// Map values
VIR.Position := Position;
VIR.NumOfKeyValuePairs := NumOfKeyValuePairs;
VIR.KeyValuePair := KeyValuePairs;

// Forward to ITC
F_ITC_SendVIR := fbITC_Manager.M_SendData(
					meChannel	:= eChannelSrc,
					mMsgType	:= E_ITC_MsgTypeConv.VISUALIZATION_INFORMATION_REPORT,
					mpData		:= ADR(VIR),
					mLen        := SIZEOF(VIR));

END_FUNCTION

// ---- 20_Product/10_BCF/11_Conv/10_Base/F_SearchPositionOfTU_Index.TcPOU
FUNCTION F_SearchPositionOfTU_Index : ST_PositionIdent
(**************************************************************************************
 * 	Application		:	BoxControl Framework
 *	Revision		:	$Revision: 464436 $
 *	Revision date	:	$Date: 2020-10-27 15:58:44 +0100 (tis, 27 okt 2020) $
 *	Last changed by	:	$Author: d7mangc $
 *	URL				:	$URL: http://almscdc.swisslog.com/repo/SWPD/Development/BoxControlFramework/20_Release/tags/R1.12.0/01_Software/BCF/BCF/JumpStart/20_Product/10_BCF/11_Conv/10_Base/F_SearchPositionOfTU_Index.TcPOU $
 *
 *	Purpose			:	Searchs for the FunctionNumber according the TU-DataIndex.
 *						
 *
 * ------------------------------------------------------------------------------------
 *	Copyright Swisslog [IP AG], Switzerland. All rights reserved.
 * 
 * ------------------------------------------------------------------------------------
 *	
 * 	Revision History: 
 *
 * 	VERSION			DATE			INITIALS			DESCRIPTION
 *	0.1				01.01.2001		swl					Example
 *
 **************************************************************************************)
VAR_INPUT
	TU_DataIndex  			: DINT; // Index variable
	eStartFunctionNumber 	: E_FunctionNumber; // Start loop from this ElementNumber 
END_VAR

VAR
	eFunctionNumber  		: E_FunctionNumber;  // Function incrementor 
	ZoneNumber				: INT; // Zone number
	FoundOnFunction			: BOOL; // Requested index was found on a function
	FoundOnZone				: BOOL; // Requested index was found on a zone
END_VAR

// Initialize
F_SearchPositionOfTU_Index.eFunctionNumber := 0;
F_SearchPositionOfTU_Index.ZoneNumber := 0;

// If no start function number is set
IF eStartFunctionNumber <= 0 THEN
	//Default set first function
	eStartFunctionNumber := F_BEGIN_FUNCTION + 1;
END_IF

// Loop through all functions
FOR eFunctionNumber := eStartFunctionNumber TO F_END_FUNCTION - 1 BY 1 DO
	// If a valid reference was found, check if a function contains on any
	// zone the requested TU Index 
	IF __ISVALIDREF(FunctionRegistry[eFunctionNumber].rFunction) THEN
		FoundOnFunction := FunctionRegistry[eFunctionNumber].rFunction.M_FindTU_DataIndex(
							mZoneNumber := 0,
							mTU_DataIndex := TU_DataIndex);

		// If the requested index could be determined on a function,
		// try to find the specific zone
		IF FoundOnFunction THEN
			// Set return value of the function	
			F_SearchPositionOfTU_Index.eFunctionNumber := eFunctionNumber;
		
			// Loop through all zones of this function 
			FOR ZoneNumber := 1 TO FunctionRegistry[eFunctionNumber].rFunction.SettingsFunction.NumberOfZones BY 1 DO
				FoundOnZone := FunctionRegistry[eFunctionNumber].rFunction.M_FindTU_DataIndex(
								mZoneNumber := ZoneNumber,
								mTU_DataIndex := TU_DataIndex);
				// Zone was found 
				IF FoundOnZone THEN
					// Set return value of the zone
					F_SearchPositionOfTU_Index.ZoneNumber := ZoneNumber;
					EXIT;
				END_IF
			END_FOR
		END_IF
		
		// If search was succesful
		IF FoundOnFunction THEN
			// Stop, and return result
			RETURN;
		END_IF
	END_IF
END_FOR

// Update position name
F_SearchPositionOfTU_Index.PositionName := F_GetFunctionName(eFunctionNumber := F_SearchPositionOfTU_Index.eFunctionNumber,
															 ZoneNumber := F_SearchPositionOfTU_Index.ZoneNumber);

END_FUNCTION

// ---- 20_Product/10_BCF/11_Conv/12_E_Functions/10_Helper/F_GetFunctionName.TcPOU
FUNCTION F_GetFunctionName : STRING(NAME_LENGTH)
(**************************************************************************************
 * 	Application		:	BoxControl Framework
 *	Revision		:	$Revision: 404529 $
 *	Revision date	:	$Date: 2018-04-23 08:21:38 +0200 (Mo., 23 Apr 2018) $
 *	Last changed by	:	$Author: b7bolm $
 *	URL				:	$URL: http://almscdc.swisslog.com/repo/SWPD/Development/BoxControlFramework/20_Release/trunk/01_Software/BCF/BCF/JumpStart/20_Product/10_App/12_E_Functions/10_Lib/10_Conv/10_Functions/F_GetFunctionName.TcPOU $
 *
 *	Purpose			:	Return function name
 *
 * ------------------------------------------------------------------------------------
 *	Copyright Swisslog [IP AG], Switzerland. All rights reserved.
 * 
 * ------------------------------------------------------------------------------------
 *	
 * 	Revision History: 
 *
 * VERSION DATE         INITIALS     DESCRIPTION
 * 0.0     DD.MM.YYYY   (name)       (explain customized modifications)
 *
 **************************************************************************************)
VAR_INPUT
	eFunctionNumber		: E_FunctionNumber; // Function number
	ZoneNumber			: INT; // Zone number
END_VAR
VAR
	DebugMsg				: T_MAXSTRING; // Debug message
END_VAR

// Check if function number is valid
IF eFunctionNumber > E_FunctionNumber.F_BEGIN_FUNCTION AND
   eFunctionNumber < E_FunctionNumber.F_END_FUNCTION THEN

	// Check reference is valid
	IF __ISVALIDREF(FunctionRegistry[eFunctionNumber].rFunction) THEN
		// If the request goes to the function
		IF ZoneNumber = 0 THEN
			// Return function name
			F_GetFunctionName := FunctionRegistry[eFunctionNumber].rFunction.SettingsFunction.FunctionName;
		ELSIF ZoneNumber > 0 AND ZoneNumber <= NUMBER_OF_ZONES_PER_FUNCTION THEN
			// Return zone name
			F_GetFunctionName := FunctionRegistry[eFunctionNumber].rFunction.SettingsFunction.Zone[ZoneNumber].ZoneName;
		ELSE
			F_GetFunctionName:= '';
			//-- debug message ------------------------------------------------
			// example: '11-000-0000-00-0,  invalid function/zone number,  function = 21,  zone = 1'
			DebugMsg:= '';
			DebugMsg:= CONCAT(DebugMsg, F_AddDividerToSisString(SubsystemRegistry.SubsystemName));
			DebugMsg:= CONCAT(DebugMsg, ',  invalid function/zone number');
			DebugMsg:= CONCAT(DebugMsg, DebugTextBlocks.FUNCTIONNBR);
			DebugMsg:= CONCAT(DebugMsg, TO_STRING(eFunctionNumber));
			DebugMsg:= CONCAT(DebugMsg, DebugTextBlocks.ZONENBR);
			DebugMsg:= CONCAT(DebugMsg, INT_TO_STRING(ZoneNumber));
			fbDebugMsgManager.M_SendMessage(meMessageType:= E_DebugMsgType.ERROR,
											mDebugSource := 'F_GetFunctionName', 
											mpMsgData    := ADR(DebugMsg),
											mMsgDataLen  := INT_TO_UDINT(LEN(DebugMsg)));
		END_IF
   END_IF
END_IF

END_FUNCTION

// ---- 20_Product/10_BCF/11_Conv/12_E_Functions/10_Helper/F_AddDividerToSisString.TcPOU
// adds '-' divider to a sis string: MMGGGEEEEFFZ -> MM-GGG-EEEE-FF-Z, even if there is already some dividers: M-M-G-G-G-E-E-E-E-F-F-Z -> MM-GGG-EEEE-FF-Z
FUNCTION PUBLIC F_AddDividerToSisString : STRING[NAME_LENGTH]

(**************************************************************************************
 * 	Application		:	BoxControl Framework
 *	Revision		:	$Revision: 461869 $
 *	Revision date	:	$Date: 2020-09-25 14:40:24 +0200 (Fr., 25 Sep 2020) $
 *	Last changed by	:	$Author: d7mangc $
 *	URL				:	$URL: http://almscdc.swisslog.com/repo/SWPD/Development/BoxControlFramework/20_Release/branches/R1.x/01_Software/BCF/BCF/JumpStart/20_Product/10_BCF/11_Conv/12_E_Functions/10_Helper/F_CreateTU_DataString.TcPOU $
 *
 *	Purpose			:	adds divider between subsystem, switchgroup, element, function and zone number
 * 						String: 'MM-GGG-EEEE-FF-Z'
 *
 * ------------------------------------------------------------------------------------
 *	Copyright Swisslog [IP AG], Switzerland. All rights reserved.
 * 
 * ------------------------------------------------------------------------------------
 *	
 * 	Revision History: 
 *
 * VERSION DATE         INITIALS     DESCRIPTION
 * 0.0     DD.MM.YYYY   (name)       (explain customized modifications)
 *
 **************************************************************************************)

//***********************************************************************************************************
VAR_INPUT
	Name				: STRING[NAME_LENGTH]		:= '';
END_VAR

//***********************************************************************************************************
VAR
	Without				: STRING[NAME_LENGTH]		:= '';
	Result				: STRING[NAME_LENGTH]		:= '';
	Src					: WORD						:= 0;
	Dst					: WORD						:= 0;
	Char				: BYTE						:= 0;
END_VAR


// initialize
memset( destAddr:= ADR(Without),  fillByte:= 16#00,  n:= SIZEOF(Without)  );
memset( destAddr:= ADR(Result),   fillByte:= 16#00,  n:= SIZEOF(Result)   );


// has name already divider? ( and remove it)
Src:= 0;
Dst:= 0;
WHILE(Name[Src] <> 16#00)DO
	Char:= Name[Src];
	Src := Src + 1;

	// valid characters?
	IF(Char >= 16#30) AND (Char <= 16#39)THEN
		Without[Dst]:= Char;
		Dst:= Dst + 1;
		CONTINUE;

	ELSIF Char >= 16#2D THEN (* '-' *)
		CONTINUE;
	END_IF

	// invalid
	F_AddDividerToSisString:= Name;
	RETURN;
END_WHILE


// add divider to specific positions
Src:= 0;
Dst:= 0;
WHILE(Without[Src] <> 16#00)DO
	// string ends
	IF Dst >= SIZEOF(Result) THEN
		Dst:= SIZEOF(Result) - 1; // make space for termination
		EXIT;
	END_IF
	
	// add divider
	IF    Src =  2 THEN  Result[Dst]:= 16#2D;  Dst:= Dst + 1;  // MM -> GGG
	ELSIF Src =  5 THEN  Result[Dst]:= 16#2D;  Dst:= Dst + 1;  // GGG -> EEEE
	ELSIF Src =  9 THEN  Result[Dst]:= 16#2D;  Dst:= Dst + 1;  // EEEE -> FF
	ELSIF Src = 11 THEN  Result[Dst]:= 16#2D;  Dst:= Dst + 1;  // FF -> Z
	END_IF
	
	// string ends
	IF Dst >= SIZEOF(Result)THEN
		Dst:= SIZEOF(Result) - 1; // make space for termination
		EXIT;
	END_IF
	
	// copy character
	Result[Dst]:= Without[Src];
	
	// continue
	Src:= Src + 1;
	Dst:= Dst + 1;
END_WHILE

Result[Dst]:= 16#00;


// done
F_AddDividerToSisString:= Result;

END_FUNCTION

// ---- 20_Product/10_BCF/11_Conv/12_E_Functions/10_Helper/F_CreateTU_DataString.TcPOU
// Creates a text string with TU data information: 'TU_DataIndex = 1979,  TuID = 0012345600,  AssignmentID = 19790109'
FUNCTION PUBLIC F_CreateTU_DataString : STRING[127]

(**************************************************************************************
 * 	Application		:	BoxControl Framework
 *	Revision		:	$Revision: 474106 $
 *	Revision date	:	$Date: 2021-03-26 07:58:15 +0100 (fre, 26 mar 2021) $
 *	Last changed by	:	$Author: d7mangc $
 *	URL				:	$URL: http://almscdc.swisslog.com/repo/SWPD/Development/BoxControlFramework/20_Release/tags/R1.12.0/01_Software/BCF/BCF/JumpStart/20_Product/10_BCF/11_Conv/12_E_Functions/10_Helper/F_CreateTU_DataString.TcPOU $
 *
 *	Purpose			:	Creates a text string with TU data information which can be used for debug messages
 * 						String: 'TU_DataIndex = 1979,  TuID = 0012345600,  AssignmentID = 19790109'
 *
 * ------------------------------------------------------------------------------------
 *	Copyright Swisslog [IP AG], Switzerland. All rights reserved.
 * 
 * ------------------------------------------------------------------------------------
 *	
 * 	Revision History: 
 *
 * VERSION DATE         INITIALS     DESCRIPTION
 * 0.0     DD.MM.YYYY   (name)       (explain customized modifications)
 *
 **************************************************************************************)
VAR_INPUT
	TU_DataIndex 	: DINT; // TU data index used to create string from
END_VAR

VAR
	TU_Data 		: ST_TU_Data;
	Result			: STRING[127];
END_VAR

// Prepaire internal vars
TU_Data := TU_Table.TU_DataTable[TU_DataIndex];
Result := '';

// TU data index
Result := CONCAT(Result, DebugTextBlocks.TU_DATA_INDEX);
Result := CONCAT(Result, DINT_TO_STRING(TU_DataIndex));

// TU ID
Result := CONCAT(Result,DebugTextBlocks.TUID);
Result := CONCAT(Result, TU_Data.TU_ID.ASCII);

// Assignment ID
Result := CONCAT(Result, DebugTextBlocks.AssignmentID);
Result := CONCAT(Result, UDINT_TO_STRING(TU_Data.AssignmentID));

// Return value
F_CreateTU_DataString := Result;

END_FUNCTION

// ---- 20_Product/10_BCF/11_Conv/10_Base/F_DeleteTU_Data.TcPOU
FUNCTION F_DeleteTU_Data : BOOL
(**************************************************************************************
 * 	Application		:	BoxControl Framework
 *	Revision		:	$Revision: 404529 $
 *	Revision date	:	$Date: 2018-04-23 08:21:38 +0200 (Mo., 23 Apr 2018) $
 *	Last changed by	:	$Author: d7mangc $
 *	URL				:	$URL: http://almscdc.swisslog.com/repo/SWPD/Development/BoxControlFramework/20_Release/trunk/01_Software/BCF/BCF/JumpStart/20_Product/10_App/10_Base/10_Lib/10_Conv/F_DeleteTU_Data.TcPOU $
 *
 *	Purpose			:	Deleting TU-Data. 
 *						Return True - Deleting was successfull
 *
 * ------------------------------------------------------------------------------------
 *	Copyright Swisslog [IP AG], Switzerland. All rights reserved.
 * 
 * ------------------------------------------------------------------------------------
 *	
 * 	Revision History: 
 *
 * VERSION DATE         INITIALS     DESCRIPTION
 * 0.0     DD.MM.YYYY   (name)       (explain customized modifications) *
 *
 **************************************************************************************)
VAR_INPUT
	TU_DataIndex				: DINT; // TU data index
	NoTTC						: BOOL; // No TTC will be sent, used for external destinations
END_VAR

VAR
	FunctionNumberOfTU_Data		: ST_PositionIdent; // Function data
	LastKnownFunctionName		: STRING(System.NAME_LENGTH); // Postion
	eFunctionNumber  			: E_FunctionNumber; // Iterator
	ZoneNumber					: INT; // Zone iterator
	IndexDeleted				: BOOL; // Deleted
	IndexWasFoundonPosition		: BOOL; // Index was found on a position
	DebugMsg					: T_MAXSTRING; // Debug msg
	TTC							: ST_ITC_TTC; // TTC
END_VAR

// Initialize
F_DeleteTU_Data := FALSE;
IndexWasFoundonPosition := FALSE;
FunctionNumberOfTU_Data.eFunctionNumber := F_BEGIN_FUNCTION;
FunctionNumberOfTU_Data.ZoneNumber := 0;

// Delete TU data only if index is valid 
IF TU_DataIndex > 0 THEN
	// Loop through all elements 
	FOR eFunctionNumber := F_BEGIN_FUNCTION + 1 TO F_END_FUNCTION - 1 BY 1 DO
		// Search FunctionNumber and ZoneIndex belonging to the TU_DataIndex 
		FunctionNumberOfTU_Data := F_SearchPositionOfTU_Index(
										TU_DataIndex 		 := TU_DataIndex, 
										eStartFunctionNumber := FunctionNumberOfTU_Data.eFunctionNumber);
		
		// Delete TU-DataIndex if it is used by a position
		IF FunctionNumberOfTU_Data.eFunctionNumber > E_FunctionNumber.F_BEGIN_FUNCTION THEN
			// Reference valid
			IF __ISVALIDREF(FunctionRegistry[FunctionNumberOfTU_Data.eFunctionNumber].rFunction) THEN
				// Remeber TU index was found on a position (For reporting)
				IndexWasFoundonPosition := TRUE;

				// Forward delete command to the function (Zone = 0) and all zones (Zone > 0)
				FOR ZoneNumber := 0 TO FunctionRegistry[FunctionNumberOfTU_Data.eFunctionNumber].rSettingsFunction.NumberOfZones DO
					// If a TU index should be deleted on a position an init command is not needed for that
					// Otherwise it is possible that we delete during a transport an Index, and after the init we delete a new index as well
					IndexDeleted := FunctionRegistry[FunctionNumberOfTU_Data.eFunctionNumber].rFunction.M_DeleteTU_DataIndex(
										mZoneNumber 	:= ZoneNumber,
										mTU_DataIndex 	:= TU_DataIndex,
										mInit			:= FALSE);
										
					// Delete executed, report it
					IF IndexDeleted THEN
						LastKnownFunctionName := F_GetFunctionName(eFunctionNumber:= FunctionNumberOfTU_Data.eFunctionNumber,
																	ZoneNumber	  := ZoneNumber);
						//-- debug message ------------------------------------------------
						// example: '11-001-1979-01-9,  TU_DataIndex deleted,  TU_DataIndex = 1979,  TuID = 0012345600,  AssignmentID = 19790109'
						DebugMsg:= '';
						DebugMsg:= CONCAT(DebugMsg, F_AddDividerToSisString(LastKnownFunctionName));
						DebugMsg:= CONCAT(DebugMsg, ',  TU_DataIndex deleted');
						DebugMsg:= CONCAT(DebugMsg, F_CreateTU_DataString(TU_DataIndex));
						fbDebugMsgManager.M_SendMessage(meMessageType:= E_DebugMsgType.INFO,
														mDebugSource := 'F_DeleteTU_Data', 
														mpMsgData    := ADR(DebugMsg),
														mMsgDataLen  := INT_TO_UDINT(LEN(DebugMsg)));
						
						// If the assignement is active notify the MFCS about the deletion 
						IF TU_DataTable[TU_DataIndex].DataSet.JobPresent AND NOT NoTTC THEN
							// Insert current position
							TTC.Position := F_ReduceToAlphaNumeric(
												InputString := FunctionRegistry[FunctionNumberOfTU_Data.eFunctionNumber].Zone[ZoneNumber].ZoneName); 					
							
							// If no position is existing take the last known position from the TU data
							IF TTC.Position = '' THEN
								TTC.Position := F_GetFunctionName(
														eFunctionNumber := TU_DataTable[TU_DataIndex].TimeStamp.eInsertFunctionNumber,
														ZoneNumber		:= TU_DataTable[TU_DataIndex].TimeStamp.InsertZoneNumber);

								// If still no position is existing take the subsystem name instead
								IF TTC.Position = '' THEN
									TTC.Position := F_ReduceToAlphaNumeric(
														InputString :=Registry.SubsystemRegistry.SubsystemName);
								END_IF	
							END_IF

							TTC.TU_DataIndex := TU_DataIndex;
							TTC.MsgSequence := 0;
							TTC.TU_ID :=  TU_DataTable[TU_DataIndex].TU_ID.ASCII;
							TTC.AssignmentID :=  TU_DataTable[TU_DataIndex].AssignmentID;
							TTC.ReturnCode := E_ErrorConv.DESTINATION_NOT_REACHABLE;
						
							System.fbITC_Manager.M_SendData(
								meChannel := 0, 
								mMsgType  := E_ITC_MsgTypeConv.TRANSPORT_TASK_COMPLETE, 
								mpData    := ADR(TTC),
								mLen	  := SIZEOF(TTC));
						END_IF
					END_IF
				END_FOR
			END_IF
		ELSE
			EXIT;
		END_IF
	END_FOR

	// If the index is not found on a position
	IF NOT IndexWasFoundonPosition THEN
		LastKnownFunctionName := F_GetFunctionName(
								eFunctionNumber := TU_DataTable[TU_DataIndex].TimeStamp.eInsertFunctionNumber,
								ZoneNumber		:= TU_DataTable[TU_DataIndex].TimeStamp.InsertZoneNumber);
		//-- debug message ------------------------------------------------
		// example: '11-001-1979-01-9,  TU_DataIndex deleted,  TU_DataIndex = 1979,  TuID = 0012345600,  AssignmentID = 19790109'
		DebugMsg:= '';
		DebugMsg:= CONCAT(DebugMsg, F_AddDividerToSisString(LastKnownFunctionName));
		DebugMsg:= CONCAT(DebugMsg, 'TU_DataIndex deleted');
		DebugMsg:= CONCAT(DebugMsg, F_CreateTU_DataString(TU_DataIndex));
		fbDebugMsgManager.M_SendMessage(meMessageType:= E_DebugMsgType.INFO,
										mDebugSource := 'F_DeleteTU_Data', 
										mpMsgData    := ADR(DebugMsg),
										mMsgDataLen  := INT_TO_UDINT(LEN(DebugMsg)));

		// If the assignement is active notify the MFCS about the deletion
		IF TU_DataTable[TU_DataIndex].DataSet.JobPresent AND NOT NoTTC THEN
			// Use the last known position from the TU data
			TTC.Position := F_ReduceToAlphaNumeric(
								InputString := LastKnownFunctionName);

			// If no position is existing take the subsystem name instead
			IF TTC.Position = '' THEN
				TTC.Position := F_ReduceToAlphaNumeric(
									InputString := Registry.SubsystemRegistry.SubsystemName);
			END_IF		

			TTC.TU_DataIndex := TU_DataIndex;
			TTC.MsgSequence := 0;
			TTC.TU_ID :=  TU_DataTable[TU_DataIndex].TU_ID.ASCII;
			TTC.AssignmentID :=  TU_DataTable[TU_DataIndex].AssignmentID;
			TTC.ReturnCode := E_ErrorConv.DESTINATION_NOT_REACHABLE;
		
			System.fbITC_Manager.M_SendData(
				meChannel := 0, 
				mMsgType  := E_ITC_MsgTypeConv.TRANSPORT_TASK_COMPLETE, 
				mpData    := ADR(TTC),
				mLen	  := SIZEOF(TTC));
		END_IF
	END_IF
	
	// Delete TU_Data set in table
	MEMSET(ADR(TU_DataTable[TU_DataIndex]), fillByte := 0, SIZEOF(TU_DataTable[TU_DataIndex]));
	// Delete successful
	F_DeleteTU_Data := TRUE;
END_IF

END_FUNCTION

// ---- 10_Project/10_App/10_Config/F_UpdateReferences.TcPOU
FUNCTION F_UpdateReferences



SubsystemRegistry.rSubsystem                                      REF= fbSubsystem10;
GroupRegistry[E_GroupNumber.G_SG_001].rGroup                      REF= fbSG_001;
ElementRegistry[E_ElementNumber.E_10_001_0200_00_0].rElement      REF= fbEL_10_001_0200_00_0;
FunctionRegistry[E_FunctionNumber.F_10_001_0200_01_0].rFunction   REF= fbF_10_001_0200_01_0;
FunctionRegistry[E_FunctionNumber.F_10_001_0200_02_0].rFunction   REF= fbF_10_001_0200_02_0;
ElementRegistry[E_ElementNumber.E_10_001_0201_00_0].rElement      REF= fbEL_10_001_0201_00_0;
FunctionRegistry[E_FunctionNumber.F_10_001_0201_01_0].rFunction   REF= fbF_10_001_0201_01_0;
ElementRegistry[E_ElementNumber.E_10_001_0202_00_0].rElement      REF= fbEL_10_001_0202_00_0;
FunctionRegistry[E_FunctionNumber.F_10_001_0202_01_0].rFunction   REF= fbF_10_001_0202_01_0;
ElementRegistry[E_ElementNumber.E_10_001_0203_00_0].rElement      REF= fbEL_10_001_0203_00_0;
FunctionRegistry[E_FunctionNumber.F_10_001_0203_01_0].rFunction   REF= fbF_10_001_0203_01_0;
FunctionRegistry[E_FunctionNumber.F_10_001_0203_02_0].rFunction   REF= fbF_10_001_0203_02_0;
FunctionRegistry[E_FunctionNumber.F_10_001_0203_03_0].rFunction   REF= fbF_10_001_0203_03_0;
FunctionRegistry[E_FunctionNumber.F_10_001_0203_04_0].rFunction   REF= fbF_10_001_0203_04_0;
FunctionRegistry[E_FunctionNumber.F_10_001_0203_05_0].rFunction   REF= fbF_10_001_0203_05_0;
ElementRegistry[E_ElementNumber.E_10_001_0204_00_0].rElement      REF= fbEL_10_001_0204_00_0;
FunctionRegistry[E_FunctionNumber.F_10_001_0204_01_0].rFunction   REF= fbF_10_001_0204_01_0;
ElementRegistry[E_ElementNumber.E_10_001_0205_00_0].rElement      REF= fbEL_10_001_0205_00_0;
ElementRegistry[E_ElementNumber.E_10_001_0207_00_0].rElement      REF= fbEL_10_001_0207_00_0;
FunctionRegistry[E_FunctionNumber.F_10_001_0207_01_0].rFunction   REF= fbF_10_001_0207_01_0;
FunctionRegistry[E_FunctionNumber.F_10_001_0207_02_0].rFunction   REF= fbF_10_001_0207_02_0;
ElementRegistry[E_ElementNumber.E_10_001_0208_00_0].rElement      REF= fbEL_10_001_0208_00_0;
FunctionRegistry[E_FunctionNumber.F_10_001_0208_01_0].rFunction   REF= fbF_10_001_0208_01_0;
ElementRegistry[E_ElementNumber.E_10_001_0209_00_0].rElement      REF= fbEL_10_001_0209_00_0;
FunctionRegistry[E_FunctionNumber.F_10_001_0209_01_0].rFunction   REF= fbF_10_001_0209_01_0;
ElementRegistry[E_ElementNumber.E_10_001_0211_00_0].rElement      REF= fbEL_10_001_0211_00_0;
FunctionRegistry[E_FunctionNumber.F_10_001_0211_01_0].rFunction   REF= fbF_10_001_0211_01_0;
ElementRegistry[E_ElementNumber.E_10_001_0212_00_0].rElement      REF= fbEL_10_001_0212_00_0;
FunctionRegistry[E_FunctionNumber.F_10_001_0212_01_0].rFunction   REF= fbF_10_001_0212_01_0;
ElementRegistry[E_ElementNumber.E_10_001_0213_00_0].rElement      REF= fbEL_10_001_0213_00_0;
FunctionRegistry[E_FunctionNumber.F_10_001_0213_01_0].rFunction   REF= fbF_10_001_0213_01_0;
FunctionRegistry[E_FunctionNumber.F_10_001_0213_02_0].rFunction   REF= fbF_10_001_0213_02_0;
ElementRegistry[E_ElementNumber.E_10_001_0214_00_0].rElement      REF= fbEL_10_001_0214_00_0;
FunctionRegistry[E_FunctionNumber.F_10_001_0214_01_0].rFunction   REF= fbF_10_001_0214_01_0;
ElementRegistry[E_ElementNumber.E_10_001_0215_00_0].rElement      REF= fbEL_10_001_0215_00_0;
FunctionRegistry[E_FunctionNumber.F_10_001_0215_01_0].rFunction   REF= fbF_10_001_0215_01_0;
FunctionRegistry[E_FunctionNumber.F_10_001_0215_02_0].rFunction   REF= fbF_10_001_0215_02_0;
FunctionRegistry[E_FunctionNumber.F_10_001_0215_03_0].rFunction   REF= fbF_10_001_0215_03_0;
ElementRegistry[E_ElementNumber.E_10_001_0216_00_0].rElement      REF= fbEL_10_001_0216_00_0;
FunctionRegistry[E_FunctionNumber.F_10_001_0216_01_0].rFunction   REF= fbF_10_001_0216_01_0;
FunctionRegistry[E_FunctionNumber.F_10_001_0216_02_0].rFunction   REF= fbF_10_001_0216_02_0;
ElementRegistry[E_ElementNumber.E_10_001_0217_00_0].rElement      REF= fbEL_10_001_0217_00_0;
FunctionRegistry[E_FunctionNumber.F_10_001_0217_01_0].rFunction   REF= fbF_10_001_0217_01_0;
ElementRegistry[E_ElementNumber.E_10_001_0218_00_0].rElement      REF= fbEL_10_001_0218_00_0;
FunctionRegistry[E_FunctionNumber.F_10_001_0218_01_0].rFunction   REF= fbF_10_001_0218_01_0;
ElementRegistry[E_ElementNumber.E_10_001_0219_00_0].rElement      REF= fbEL_10_001_0219_00_0;
FunctionRegistry[E_FunctionNumber.F_10_001_0219_01_0].rFunction   REF= fbF_10_001_0219_01_0;
ElementRegistry[E_ElementNumber.E_10_001_0220_00_0].rElement      REF= fbEL_10_001_0220_00_0;
FunctionRegistry[E_FunctionNumber.F_10_001_0220_01_0].rFunction   REF= fbF_10_001_0220_01_0;
ElementRegistry[E_ElementNumber.E_10_001_0221_00_0].rElement      REF= fbEL_10_001_0221_00_0;
FunctionRegistry[E_FunctionNumber.F_10_001_0221_01_0].rFunction   REF= fbF_10_001_0221_01_0;
ElementRegistry[E_ElementNumber.E_10_001_0222_00_0].rElement      REF= fbEL_10_001_0222_00_0;
FunctionRegistry[E_FunctionNumber.F_10_001_0222_01_0].rFunction   REF= fbF_10_001_0222_01_0;
ElementRegistry[E_ElementNumber.E_10_001_0223_00_0].rElement      REF= fbEL_10_001_0223_00_0;
ElementRegistry[E_ElementNumber.E_10_001_0225_00_0].rElement      REF= fbEL_10_001_0225_00_0;
FunctionRegistry[E_FunctionNumber.F_10_001_0225_01_0].rFunction   REF= fbF_10_001_0225_01_0;
ElementRegistry[E_ElementNumber.E_10_001_0226_00_0].rElement      REF= fbEL_10_001_0226_00_0;
FunctionRegistry[E_FunctionNumber.F_10_001_0226_01_0].rFunction   REF= fbF_10_001_0226_01_0;
ElementRegistry[E_ElementNumber.E_10_001_0227_00_0].rElement      REF= fbEL_10_001_0227_00_0;
FunctionRegistry[E_FunctionNumber.F_10_001_0227_01_0].rFunction   REF= fbF_10_001_0227_01_0;
ElementRegistry[E_ElementNumber.E_10_001_0230_00_0].rElement      REF= fbEL_10_001_0230_00_0;
FunctionRegistry[E_FunctionNumber.F_10_001_0230_01_0].rFunction   REF= fbF_10_001_0230_01_0;
ElementRegistry[E_ElementNumber.E_10_001_0232_00_0].rElement      REF= fbEL_10_001_0232_00_0;
FunctionRegistry[E_FunctionNumber.F_10_001_0232_01_0].rFunction   REF= fbF_10_001_0232_01_0;
FunctionRegistry[E_FunctionNumber.F_10_001_0232_02_0].rFunction   REF= fbF_10_001_0232_02_0;
ElementRegistry[E_ElementNumber.E_10_001_0233_00_0].rElement      REF= fbEL_10_001_0233_00_0;
FunctionRegistry[E_FunctionNumber.F_10_001_0233_01_0].rFunction   REF= fbF_10_001_0233_01_0;
GroupRegistry[E_GroupNumber.G_SG_002].rGroup                      REF= fbSG_002;
ElementRegistry[E_ElementNumber.E_10_002_0206_00_0].rElement      REF= fbEL_10_002_0206_00_0;
FunctionRegistry[E_FunctionNumber.F_10_002_0206_01_0].rFunction   REF= fbF_10_002_0206_01_0;

END_FUNCTION

// ---- 10_Project/10_App/10_Config/F_UpdateISR.TcPOU
FUNCTION F_UpdateISR



ISR_SignalType[2].SignalNumber[0001] :=  fbF_10_001_0200_01_0.ZoneData[1].TransportControlData.NumberOfPresentTUs > 0;
ISR_SignalType[2].SignalNumber[0002] :=  fbF_10_001_0201_01_0.ZoneData[1].TransportControlData.NumberOfPresentTUs > 0;
ISR_SignalType[2].SignalNumber[0003] :=  fbF_10_001_0202_01_0.ZoneData[1].TransportControlData.NumberOfPresentTUs > 0;
ISR_SignalType[2].SignalNumber[0004] :=  fbF_10_001_0203_01_0.ZoneData[1].TransportControlData.NumberOfPresentTUs > 0;
ISR_SignalType[2].SignalNumber[0005] :=  fbF_10_001_0204_01_0.ZoneData[1].TransportControlData.NumberOfPresentTUs > 0;
ISR_SignalType[2].SignalNumber[0006] :=  fbF_10_001_0207_01_0.ZoneData[1].TransportControlData.NumberOfPresentTUs > 0;
ISR_SignalType[2].SignalNumber[0007] :=  fbF_10_001_0208_01_0.ZoneData[1].TransportControlData.NumberOfPresentTUs > 0;
ISR_SignalType[2].SignalNumber[0008] :=  fbF_10_001_0209_01_0.ZoneData[1].TransportControlData.NumberOfPresentTUs > 0;
ISR_SignalType[2].SignalNumber[0009] :=  fbF_10_001_0211_01_0.ZoneData[1].TransportControlData.NumberOfPresentTUs > 0;
ISR_SignalType[2].SignalNumber[0010] :=  fbF_10_001_0212_01_0.ZoneData[1].TransportControlData.NumberOfPresentTUs > 0;
ISR_SignalType[2].SignalNumber[0011] :=  fbF_10_001_0213_01_0.ZoneData[1].TransportControlData.NumberOfPresentTUs > 0;
ISR_SignalType[2].SignalNumber[0012] :=  fbF_10_001_0214_01_0.ZoneData[1].TransportControlData.NumberOfPresentTUs > 0;
ISR_SignalType[2].SignalNumber[0013] :=  fbF_10_001_0215_01_0.ZoneData[1].TransportControlData.NumberOfPresentTUs > 0;
ISR_SignalType[2].SignalNumber[0014] :=  fbF_10_001_0215_02_0.ZoneData[1].TransportControlData.NumberOfPresentTUs > 0;
ISR_SignalType[2].SignalNumber[0015] :=  fbF_10_001_0216_01_0.ZoneData[1].TransportControlData.NumberOfPresentTUs > 0;
ISR_SignalType[2].SignalNumber[0016] :=  fbF_10_001_0216_01_0.ZoneData[2].TransportControlData.NumberOfPresentTUs > 0;
ISR_SignalType[2].SignalNumber[0017] :=  fbF_10_001_0217_01_0.ZoneData[1].TransportControlData.NumberOfPresentTUs > 0;
ISR_SignalType[2].SignalNumber[0018] :=  fbF_10_001_0218_01_0.ZoneData[1].TransportControlData.NumberOfPresentTUs > 0;
ISR_SignalType[2].SignalNumber[0019] :=  fbF_10_001_0218_01_0.ZoneData[2].TransportControlData.NumberOfPresentTUs > 0;
ISR_SignalType[2].SignalNumber[0020] :=  fbF_10_001_0219_01_0.ZoneData[1].TransportControlData.NumberOfPresentTUs > 0;
ISR_SignalType[2].SignalNumber[0021] :=  fbF_10_001_0219_01_0.ZoneData[2].TransportControlData.NumberOfPresentTUs > 0;
ISR_SignalType[2].SignalNumber[0022] :=  fbF_10_001_0220_01_0.ZoneData[1].TransportControlData.NumberOfPresentTUs > 0;
ISR_SignalType[2].SignalNumber[0023] :=  fbF_10_001_0221_01_0.ZoneData[1].TransportControlData.NumberOfPresentTUs > 0;
ISR_SignalType[2].SignalNumber[0024] :=  fbF_10_001_0222_01_0.ZoneData[1].TransportControlData.NumberOfPresentTUs > 0;
ISR_SignalType[2].SignalNumber[0025] :=  fbF_10_001_0225_01_0.ZoneData[1].TransportControlData.NumberOfPresentTUs > 0;
ISR_SignalType[2].SignalNumber[0026] :=  fbF_10_001_0225_01_0.ZoneData[2].TransportControlData.NumberOfPresentTUs > 0;
ISR_SignalType[2].SignalNumber[0027] :=  fbF_10_001_0226_01_0.ZoneData[1].TransportControlData.NumberOfPresentTUs > 0;
ISR_SignalType[2].SignalNumber[0028] :=  fbF_10_001_0226_01_0.ZoneData[2].TransportControlData.NumberOfPresentTUs > 0;
ISR_SignalType[2].SignalNumber[0029] :=  fbF_10_001_0227_01_0.ZoneData[1].TransportControlData.NumberOfPresentTUs > 0;
ISR_SignalType[2].SignalNumber[0030] :=  fbF_10_001_0230_01_0.ZoneData[1].TransportControlData.NumberOfPresentTUs > 0;
ISR_SignalType[2].SignalNumber[0031] :=  fbF_10_001_0232_01_0.ZoneData[1].TransportControlData.NumberOfPresentTUs > 0;
ISR_SignalType[2].SignalNumber[0032] :=  fbF_10_001_0232_01_0.ZoneData[2].TransportControlData.NumberOfPresentTUs > 0;
ISR_SignalType[2].SignalNumber[0033] :=  fbF_10_001_0233_01_0.ZoneData[1].TransportControlData.NumberOfPresentTUs > 0;
ISR_SignalType[2].SignalNumber[0034] :=  fbF_10_002_0206_01_0.ZoneData[1].TransportControlData.NumberOfPresentTUs > 0;

END_FUNCTION

// ---- 20_Product/10_BCF/11_Conv/15_Subsystem/10_Helper/F_GetSubsystemOperationState.TcPOU
FUNCTION F_GetSubsystemOperationState : ST_PositionState
(**************************************************************************************
 * 	Application		:	BoxControl Framework
 *	Revision		:	$Revision: 404529 $
 *	Revision date	:	$Date: 2018-04-23 08:21:38 +0200 (Mo., 23 Apr 2018) $
 *	Last changed by	:	$Author: b7bolm $
 *	URL				:	$URL: http://almscdc.swisslog.com/repo/SWPD/Development/BoxControlFramework/20_Release/trunk/01_Software/BCF/BCF/JumpStart/20_Product/10_App/15_Subsystem/10_Lib/10_Conv/10_Functions/F_GetSubsystemOperationState.TcPOU $
 *
 *	Purpose			:	Returns group states
 *
 * ------------------------------------------------------------------------------------
 *	Copyright Swisslog [IP AG], Switzerland. All rights reserved.
 * 
 * ------------------------------------------------------------------------------------
 *	
 * 	Revision History: 
 *
 * 	VERSION			DATE			INITIALS			DESCRIPTION
 *	0.1				01.01.2001		swl					Example
 *
 **************************************************************************************)



// Get Master speed from subsystem
IF __ISVALIDREF(SubsystemRegistry.rSubsystemData) THEN
	// Return Subsystem state
	F_GetSubsystemOperationState := SubsystemRegistry.rSubsystemData.OperationState;
END_IF

END_FUNCTION

// ---- 10_Project/10_App/10_Config/F_ConfigProduct.TcPOU
FUNCTION F_ConfigProduct : BOOL



(****************************************************************************************
   Message handler
*****************************************************************************************)
fbDebugMsgManager.EnableErrors              :=TRUE;
fbDebugMsgManager.EnableInfos               :=TRUE;
fbDebugMsgManager.EnableWarnings            :=TRUE;

fbDebugMsgManager.FileHandler.MaxFileSizeKB :=4096;
fbDebugMsgManager.FileHandler.Folder        :='C:\Temp\Traces';
fbDebugMsgManager.FileHandler.Enable        :=FALSE;

(****************************************************************************************
   Configuration Product
*****************************************************************************************)
fbITC_Manager                               := fb_PB_ITC_ManagerConveyor;
fb_PB_ITC_ManagerConveyor.Config.SDI_Limit  := 0; //Limit usage of SDI's

(****************************************************************************************
   Define MFCS channels (e.g.SIS channels)
*****************************************************************************************)
fbMFCS_Channel[E_MFCS_Channel.AM] 			:= fbMFCS_SIS_AM;
fbMFCS_Channel[E_MFCS_Channel.SPOC]			:= fbMFCS_SIS_SPOC;
fbMFCS_Channel[E_MFCS_Channel.LOGGING]		:= fbMFCS_LOG;

END_FUNCTION

// ---- 10_Project/10_App/10_Config/F_ConfigCommunication.TcPOU
FUNCTION F_ConfigCommunication : BOOL
VAR
	///Set to true when connected to SynQ
	SynQComm: BOOL := FALSE;
END_VAR



(**************************************************************************************************************
   Configuration DebugMsgManager
***************************************************************************************************************)
fbDebugMsgManager.Config.SystemNumber := 10;

fbDebugMsgManager.Config.TCP_Driver.ChannelName                     := 'Debug Message Manager';
fbDebugMsgManager.Config.TCP_Driver.EnableConnection                := TRUE;
fbDebugMsgManager.Config.TCP_Driver.RemoteHost                      := '0.0.0.0';
fbDebugMsgManager.Config.TCP_Driver.RemotePort                      := 0;
fbDebugMsgManager.Config.TCP_Driver.LocalHost                       := '0.0.0.0';
fbDebugMsgManager.Config.TCP_Driver.LocalPort                       := 5000;
fbDebugMsgManager.Config.TCP_Driver.Server                          := TRUE;
fbDebugMsgManager.Config.TCP_Driver.ConnectTimeout                  := T#10S;
fbDebugMsgManager.Config.TCP_Driver.ClientRetryInterval             := T#5S;
fbDebugMsgManager.Config.TCP_Driver.ServerRetryInterval             := T#1S;
fbDebugMsgManager.Config.TCP_Driver.AcceptPollInterval              := T#10S;
fbDebugMsgManager.Config.TCP_Driver.EnableDebugMsg                  := FALSE;

(******************* Communication Parameters for SIS Engine to AM **************************)

fbMFCS_SIS_AM.Config.BaseDriver.TCP_Driver.ChannelName              := 'AM TCP/IP Driver';
fbMFCS_SIS_AM.Config.BaseDriver.TCP_Driver.EnableConnection         := TRUE;
IF SynQComm THEN
	(***Config Communication parameters when connected TO SynQ, inhuse tests(Project specific)***)  
	fbMFCS_SIS_AM.Config.BaseDriver.TCP_Driver.RemoteHost               := '10.49.134.93';
	fbMFCS_SIS_AM.Config.BaseDriver.TCP_Driver.RemotePort               := 10001;
	fbMFCS_SIS_AM.Config.BaseDriver.TCP_Driver.LocalHost                := '0.0.0.0';
	fbMFCS_SIS_AM.Config.BaseDriver.TCP_Driver.LocalPort                := 0;
	fbMFCS_SIS_AM.Config.BaseDriver.TCP_Driver.Server                   := FALSE;
ELSE
(***Config Communication parameters when connected to ComTool, stand alone tests***)  	
	fbMFCS_SIS_AM.Config.BaseDriver.TCP_Driver.RemoteHost               := '0.0.0.0';
	fbMFCS_SIS_AM.Config.BaseDriver.TCP_Driver.RemotePort               := 0;
	fbMFCS_SIS_AM.Config.BaseDriver.TCP_Driver.LocalHost                := '0.0.0.0';
	fbMFCS_SIS_AM.Config.BaseDriver.TCP_Driver.LocalPort                := 2111;
	fbMFCS_SIS_AM.Config.BaseDriver.TCP_Driver.Server                   := TRUE;	
END_IF
fbMFCS_SIS_AM.Config.BaseDriver.TCP_Driver.ConnectTimeout           := T#10S;
fbMFCS_SIS_AM.Config.BaseDriver.TCP_Driver.ClientRetryInterval      := T#5S;
fbMFCS_SIS_AM.Config.BaseDriver.TCP_Driver.ServerRetryInterval      := T#1S;
fbMFCS_SIS_AM.Config.BaseDriver.TCP_Driver.AcceptPollInterval       := T#10S;
fbMFCS_SIS_AM.Config.BaseDriver.TCP_Driver.EnableDebugMsg           := FALSE;

fbMFCS_SIS_AM.Config.BaseDriver.StartChar                           := '<';
fbMFCS_SIS_AM.Config.BaseDriver.EndChar                             := '>';
IF SynQComm THEN
(***Config Communication parameters when connected to SynQ, inhuse tests(Project spesific)***) 
	fbMFCS_SIS_AM.Config.BaseDriver.StationName                         := 'PFA_10';
	fbMFCS_SIS_AM.Config.BaseDriver.PartnerName                         := 'MOVE01';
ELSE
(***Config Communication parameters when connected to ComTool, stand alone tests***)  
	fbMFCS_SIS_AM.Config.BaseDriver.StationName                         := 'LGCS10';
	fbMFCS_SIS_AM.Config.BaseDriver.PartnerName                         := 'MOVE01';
END_IF
fbMFCS_SIS_AM.Config.BaseDriver.DoAutoSync                          := TRUE;
fbMFCS_SIS_AM.Config.BaseDriver.EnableDebugMsg                      := FALSE;
fbMFCS_SIS_AM.Config.BaseDriver.EnableBufferOverwrite               := FALSE;

fbMFCS_SIS_AM.Config.MFCS_Channel                                   := E_MFCS_Channel.AM;
fbMFCS_SIS_AM.Config.BufferLevelWarning                             := 700;
fbMFCS_SIS_AM.Config.BufferLevelAlarm                               := 900;
fbMFCS_SIS_AM.Config.MirrorChannel                                  := E_MFCS_Channel.LOGGING;

fbMFCS_SIS_AM.Config.Telegrams.SendFCR                              := FALSE;
fbMFCS_SIS_AM.Config.Telegrams.SendFSR                              := FALSE;
fbMFCS_SIS_AM.Config.Telegrams.SendECR                              := FALSE;
fbMFCS_SIS_AM.Config.Telegrams.SendESR                              := FALSE;
fbMFCS_SIS_AM.Config.Telegrams.SendGCR                              := FALSE;
fbMFCS_SIS_AM.Config.Telegrams.SendGSR                              := FALSE;
fbMFCS_SIS_AM.Config.Telegrams.SendSCR                              := FALSE;
fbMFCS_SIS_AM.Config.Telegrams.SendSSR                              := FALSE;
fbMFCS_SIS_AM.Config.Telegrams.SendMCR                              := FALSE;
fbMFCS_SIS_AM.Config.Telegrams.SendGVR                              := FALSE;
fbMFCS_SIS_AM.Config.Telegrams.SendIPR                              := TRUE;
fbMFCS_SIS_AM.Config.Telegrams.SendMSG                              := TRUE;
fbMFCS_SIS_AM.Config.Telegrams.SendPOR                              := TRUE;
fbMFCS_SIS_AM.Config.Telegrams.SendSDI                              := FALSE;
fbMFCS_SIS_AM.Config.Telegrams.SendSIR                              := FALSE;
fbMFCS_SIS_AM.Config.Telegrams.SendSNR                              := TRUE;
fbMFCS_SIS_AM.Config.Telegrams.SendTDR                              := TRUE;
fbMFCS_SIS_AM.Config.Telegrams.SendTTC                              := TRUE;
fbMFCS_SIS_AM.Config.Telegrams.SendTTQ                              := TRUE;
fbMFCS_SIS_AM.Config.Telegrams.SendTUR                              := TRUE;
fbMFCS_SIS_AM.Config.Telegrams.SendATR                              := TRUE;
fbMFCS_SIS_AM.Config.Telegrams.SendRTR                              := TRUE;
fbMFCS_SIS_AM.Config.Telegrams.SendERR                              := TRUE;
fbMFCS_SIS_AM.Config.Telegrams.SendRDR                              := TRUE;
fbMFCS_SIS_AM.Config.Telegrams.SendRAC                              := TRUE;
fbMFCS_SIS_AM.Config.Telegrams.SendVIR                              := FALSE;

(******************* Communication Parameters for SIS Engine to SPOC ************************)

fbMFCS_SIS_SPOC.Config.BaseDriver.TCP_Driver.ChannelName            := 'SPOC TCP/IP Driver';
fbMFCS_SIS_SPOC.Config.BaseDriver.TCP_Driver.EnableConnection       := TRUE;
IF SynQComm THEN
(***Config Communication parameters when connected to SynQ, inhuse tests(Project spesific)***) 
	fbMFCS_SIS_SPOC.Config.BaseDriver.TCP_Driver.RemoteHost             := '10.49.134.93';
	fbMFCS_SIS_SPOC.Config.BaseDriver.TCP_Driver.RemotePort             := 10002;
	fbMFCS_SIS_SPOC.Config.BaseDriver.TCP_Driver.LocalHost              := '0.0.0.0';
	fbMFCS_SIS_SPOC.Config.BaseDriver.TCP_Driver.LocalPort              := 0;
	fbMFCS_SIS_SPOC.Config.BaseDriver.TCP_Driver.Server                 := FALSE;
ELSE
(***Config Communication parameters when connected to ComTool, stand alone tests***)  	
	fbMFCS_SIS_SPOC.Config.BaseDriver.TCP_Driver.RemoteHost             := '0.0.0.0';
	fbMFCS_SIS_SPOC.Config.BaseDriver.TCP_Driver.RemotePort             := 0;
	fbMFCS_SIS_SPOC.Config.BaseDriver.TCP_Driver.LocalHost              := '127.0.0.1';
	fbMFCS_SIS_SPOC.Config.BaseDriver.TCP_Driver.LocalPort              := 2211;
	fbMFCS_SIS_SPOC.Config.BaseDriver.TCP_Driver.Server                 := TRUE;
END_IF
fbMFCS_SIS_SPOC.Config.BaseDriver.TCP_Driver.ConnectTimeout         := T#10S;
fbMFCS_SIS_SPOC.Config.BaseDriver.TCP_Driver.ClientRetryInterval    := T#5S;
fbMFCS_SIS_SPOC.Config.BaseDriver.TCP_Driver.ServerRetryInterval    := T#1S;
fbMFCS_SIS_SPOC.Config.BaseDriver.TCP_Driver.AcceptPollInterval	    := T#10S;
fbMFCS_SIS_SPOC.Config.BaseDriver.TCP_Driver.EnableDebugMsg	        := FALSE;

fbMFCS_SIS_SPOC.Config.BaseDriver.StartChar	                        := '<';
fbMFCS_SIS_SPOC.Config.BaseDriver.EndChar                           := '>';
IF SynQComm THEN
(***Config Communication parameters when connected to SynQ, inhuse tests(Project spesific)***) 
	fbMFCS_SIS_SPOC.Config.BaseDriver.StationName                       := 'PFA_10';
	fbMFCS_SIS_SPOC.Config.BaseDriver.PartnerName                       := 'VISU02';
ELSE
(***Config Communication parameters when connected to ComTool, stand alone tests***) 
	fbMFCS_SIS_SPOC.Config.BaseDriver.StationName                       := 'LGCS10';
	fbMFCS_SIS_SPOC.Config.BaseDriver.PartnerName                       := 'SPOC02';
END_IF
fbMFCS_SIS_SPOC.Config.BaseDriver.DoAutoSync                        := TRUE;
fbMFCS_SIS_SPOC.Config.BaseDriver.EnableDebugMsg                    := FALSE;
fbMFCS_SIS_SPOC.Config.BaseDriver.EnableBufferOverwrite             := TRUE;

fbMFCS_SIS_SPOC.Config.MFCS_Channel                                 := E_MFCS_Channel.SPOC;
fbMFCS_SIS_SPOC.Config.BufferLevelWarning                           := 700;
fbMFCS_SIS_SPOC.Config.BufferLevelAlarm                             := 900;
fbMFCS_SIS_SPOC.Config.MirrorChannel                                := E_MFCS_Channel.LOGGING;

fbMFCS_SIS_SPOC.Config.Telegrams.SendFCR                            := TRUE;
fbMFCS_SIS_SPOC.Config.Telegrams.SendFSR                            := TRUE;
fbMFCS_SIS_SPOC.Config.Telegrams.SendECR                            := TRUE;
fbMFCS_SIS_SPOC.Config.Telegrams.SendESR                            := TRUE;
fbMFCS_SIS_SPOC.Config.Telegrams.SendGCR                            := TRUE;
fbMFCS_SIS_SPOC.Config.Telegrams.SendGSR                            := TRUE;
fbMFCS_SIS_SPOC.Config.Telegrams.SendSCR                            := TRUE;
fbMFCS_SIS_SPOC.Config.Telegrams.SendSSR                            := TRUE;
fbMFCS_SIS_SPOC.Config.Telegrams.SendMCR                            := TRUE;
fbMFCS_SIS_SPOC.Config.Telegrams.SendGVR                            := TRUE;
fbMFCS_SIS_SPOC.Config.Telegrams.SendIPR                            := FALSE;
fbMFCS_SIS_SPOC.Config.Telegrams.SendMSG                            := TRUE;
fbMFCS_SIS_SPOC.Config.Telegrams.SendPOR                            := FALSE;
fbMFCS_SIS_SPOC.Config.Telegrams.SendSDI                            := FALSE;
fbMFCS_SIS_SPOC.Config.Telegrams.SendSIR                            := TRUE;
fbMFCS_SIS_SPOC.Config.Telegrams.SendSNR                            := FALSE;
fbMFCS_SIS_SPOC.Config.Telegrams.SendTDR                            := TRUE;
fbMFCS_SIS_SPOC.Config.Telegrams.SendTTC                            := FALSE;
fbMFCS_SIS_SPOC.Config.Telegrams.SendTTQ                            := FALSE;
fbMFCS_SIS_SPOC.Config.Telegrams.SendTUR                            := TRUE;
fbMFCS_SIS_SPOC.Config.Telegrams.SendATR                            := TRUE;
fbMFCS_SIS_SPOC.Config.Telegrams.SendRTR                            := TRUE;
fbMFCS_SIS_SPOC.Config.Telegrams.SendERR                            := TRUE;
fbMFCS_SIS_SPOC.Config.Telegrams.SendRDR                            := TRUE;
fbMFCS_SIS_SPOC.Config.Telegrams.SendRAC                            := FALSE;
fbMFCS_SIS_SPOC.Config.Telegrams.SendVIR                            := TRUE;
fbMFCS_SIS_SPOC.Config.Telegrams.SendISR                            := TRUE;


(******************* Communication Parameters for SIS Engine to LOG ************************)
fbMFCS_LOG.Config.BaseDriver.TCP_Driver.ChannelName                 := 'SIS log';
fbMFCS_LOG.Config.BaseDriver.TCP_Driver.EnableConnection            := TRUE;
fbMFCS_LOG.Config.BaseDriver.TCP_Driver.RemoteHost                  := '0.0.0.0';
fbMFCS_LOG.Config.BaseDriver.TCP_Driver.RemotePort                  := 0;
fbMFCS_LOG.Config.BaseDriver.TCP_Driver.LocalHost                   := '0.0.0.0';
fbMFCS_LOG.Config.BaseDriver.TCP_Driver.LocalPort                   := 6000;
fbMFCS_LOG.Config.BaseDriver.TCP_Driver.Server                      := TRUE;
fbMFCS_LOG.Config.BaseDriver.TCP_Driver.ConnectTimeout              := T#10S;
fbMFCS_LOG.Config.BaseDriver.TCP_Driver.ClientRetryInterval         := T#5S;
fbMFCS_LOG.Config.BaseDriver.TCP_Driver.ServerRetryInterval         := T#1S;
fbMFCS_LOG.Config.BaseDriver.TCP_Driver.AcceptPollInterval          := T#10S;
fbMFCS_LOG.Config.BaseDriver.TCP_Driver.EnableDebugMsg              := FALSE;

fbMFCS_LOG.Config.BaseDriver.StartChar                              := '<';
fbMFCS_LOG.Config.BaseDriver.EndChar                                := '>';
fbMFCS_LOG.Config.BaseDriver.StationName                            := 'LGCS10';
fbMFCS_LOG.Config.BaseDriver.PartnerName                            := 'SISLOG';
fbMFCS_LOG.Config.BaseDriver.DoAutoSync	                            := TRUE;
fbMFCS_LOG.Config.BaseDriver.EnableDebugMsg	                        := FALSE;
fbMFCS_LOG.Config.BaseDriver.EnableBufferOverwrite                  := TRUE;

fbMFCS_LOG.Config.MFCS_Channel                                      := E_MFCS_Channel.LOGGING;
fbMFCS_LOG.Config.BufferLevelWarning                                := 700;
fbMFCS_LOG.Config.BufferLevelAlarm                                  := 900;
fbMFCS_LOG.Config.MirrorChannel                                     := E_MFCS_Channel.BEGIN_CHANNEL;

END_FUNCTION

// ---- 10_Project/10_App/10_Config/F_ConfigPosition.TcPOU
FUNCTION F_ConfigPosition



F_ConfigPosition_001();

F_ConfigPosition_002();

END_FUNCTION

// ---- 10_Project/10_App/10_Config/F_ConfigPosition_001.TcPOU
FUNCTION F_ConfigPosition_001



(****************************** 10-001-0200-00-0 ************************************)
(*************************** ProBoxElement with one Motor *******************************)
// Configuration element 
fbEL_10_001_0200_00_0.ConfigElement.ElementName                     := '10-001-0200-00-0'; // Element name 
fbEL_10_001_0200_00_0.ConfigElement.eElementNumber                  := E_10_001_0200_00_0; // Number of the element 
fbEL_10_001_0200_00_0.ConfigElement.eSlaveElementNumber_34          := E_ElementNumber.E_BEGIN_ELEMENT; // Link from Master to slave element
fbEL_10_001_0200_00_0.ConfigElement.eElementType                    := E_ElementType.NO_TYPE; // No specific type

// Register element 
ElementRegistry[E_10_001_0200_00_0].Enable                          := TRUE; // Object is called
ElementRegistry[E_10_001_0200_00_0].eElementNumber                  := fbEL_10_001_0200_00_0.ConfigElement.eElementNumber; 

(****************************** 10-001-0200-01-0 ************************************)
(************************** ProBox Straight Transport *******************************)
// Configuration function
fbF_10_001_0200_01_0.ConfigFunction.FunctionName                       := '10-001-0200-01-0'; // Function name
fbF_10_001_0200_01_0.ConfigFunction.eFunctionNumber                    := F_10_001_0200_01_0; // Number of the function
fbF_10_001_0200_01_0.ConfigFunction.eElementLink                       := E_ElementNumber.E_10_001_0200_00_0;
fbF_10_001_0200_01_0.ConfigFunction.FunctionLink.eFunctionNumber       := E_FunctionNumber.F_BEGIN_FUNCTION;
fbF_10_001_0200_01_0.ConfigFunction.FunctionLink.ZoneNumber            := 0;
fbF_10_001_0200_01_0.ConfigFunction.eAdjacentFunctionNumberSide[1]     := E_FunctionNumber.F_BEGIN_FUNCTION;
fbF_10_001_0200_01_0.ConfigFunction.eAdjacentFunctionNumberSide[2]     := E_FunctionNumber.F_10_001_0201_01_0;
fbF_10_001_0200_01_0.ConfigFunction.ePrevFunctionNumber                := E_FunctionNumber.F_BEGIN_FUNCTION;
fbF_10_001_0200_01_0.ConfigFunction.eNextFunctionNumber                := E_FunctionNumber.F_10_001_0201_01_0;
fbF_10_001_0200_01_0.ConfigFunction.NumberOfZones                      := 1;
//Config zone 1
fbF_10_001_0200_01_0.ConfigFunction.Zone[1].ZoneName                   := '10-001-0200-01-1';
fbF_10_001_0200_01_0.ConfigFunction.Zone[1].EnableMFC                  := TRUE;
fbF_10_001_0200_01_0.ConfigFunction.Zone[1].EnableSimultaneousTransport:= FALSE; //Disable Simultaneous transport for multi zone functions
fbF_10_001_0200_01_0.ConfigFunction.Zone[1].EnableLatchOccupiedState   := TRUE;
fbF_10_001_0200_01_0.ConfigFunction.Zone[1].Length[1]                  := INT_TO_UINT(2000 / fbF_10_001_0200_01_0.ConfigFunction.NumberOfZones);	//Zone length (ie element length / number of zones)

// Register function
FunctionRegistry[F_10_001_0200_01_0].Enable                            := TRUE; (* Function will be called *)
FunctionRegistry[F_10_001_0200_01_0].eFunctionNumber                   := fbF_10_001_0200_01_0.ConfigFunction.eFunctionNumber; // Registration number


(****************************** 10-001-0200-02-0 ************************************)
(********************************* In/Out Feed ****************************************)
// Configuration function 
fbF_10_001_0200_02_0.ConfigFunction.FunctionName                     := '10-001-0200-02-0'; (* Function name *)
fbF_10_001_0200_02_0.ConfigFunction.eFunctionNumber                  := F_10_001_0200_02_0; (* Number of the function *)
fbF_10_001_0200_02_0.ConfigFunction.eElementLink                     := E_ElementNumber.E_10_001_0200_00_0; 
fbF_10_001_0200_02_0.ConfigFunction.FunctionLink.eFunctionNumber     := E_FunctionNumber.F_10_001_0200_01_0;	//Addon link to function, this is auto generated, an may need to be changed.
fbF_10_001_0200_02_0.ConfigFunction.FunctionLink.ZoneNumber          := 1;		

fbF_10_001_0200_02_0.Config.tFTLClearTime                  		  := T#5S; //Fork Truck Lift clear time
fbF_10_001_0200_02_0.Config.tTUSensorTime					  		  := T#5S; //Sensor occupied Time when to add or remove TU
fbF_10_001_0200_02_0.Config.TimeoutValueLift					  	  := T#10S; //Timeout value for lifting
fbF_10_001_0200_02_0.Config.LiftEnabled					  	  	  := FALSE; //Config if function has lift

// Register function 
FunctionRegistry[F_10_001_0200_02_0].Enable                           := TRUE; (* Function will be called *)
FunctionRegistry[F_10_001_0200_02_0].eFunctionNumber                  := fbF_10_001_0200_02_0.ConfigFunction.eFunctionNumber; (* Registration number *)


(****************************** 10-001-0201-00-0 ************************************)
(*************************** ProBoxElement with one Motor *******************************)
// Configuration element 
fbEL_10_001_0201_00_0.ConfigElement.ElementName                     := '10-001-0201-00-0'; // Element name 
fbEL_10_001_0201_00_0.ConfigElement.eElementNumber                  := E_10_001_0201_00_0; // Number of the element 
fbEL_10_001_0201_00_0.ConfigElement.eSlaveElementNumber_34          := E_ElementNumber.E_BEGIN_ELEMENT; // Link from Master to slave element
fbEL_10_001_0201_00_0.ConfigElement.eElementType                    := E_ElementType.NO_TYPE; // No specific type

// Register element 
ElementRegistry[E_10_001_0201_00_0].Enable                          := TRUE; // Object is called
ElementRegistry[E_10_001_0201_00_0].eElementNumber                  := fbEL_10_001_0201_00_0.ConfigElement.eElementNumber; 

(****************************** 10-001-0201-01-0 ************************************)
(******************************** LowLiftUnit  ***************************************)
// Configuration function
fbF_10_001_0201_01_0.ConfigFunction.FunctionName                      := '10-001-0201-01-0'; // Function name
fbF_10_001_0201_01_0.ConfigFunction.eFunctionNumber                   := F_10_001_0201_01_0; // Number of the function
fbF_10_001_0201_01_0.ConfigFunction.eElementLink                      := E_ElementNumber.E_10_001_0201_00_0;
fbF_10_001_0201_01_0.ConfigFunction.FunctionLink.eFunctionNumber      := E_FunctionNumber.F_BEGIN_FUNCTION;
fbF_10_001_0201_01_0.ConfigFunction.FunctionLink.ZoneNumber           := 0;
fbF_10_001_0201_01_0.ConfigFunction.eAdjacentFunctionNumberSide[1]    := E_FunctionNumber.F_10_001_0200_01_0;
fbF_10_001_0201_01_0.ConfigFunction.eAdjacentFunctionNumberSide[2]    := E_FunctionNumber.F_10_001_0202_01_0;
fbF_10_001_0201_01_0.ConfigFunction.ePrevFunctionNumber               := E_FunctionNumber.F_10_001_0200_01_0;
fbF_10_001_0201_01_0.ConfigFunction.eNextFunctionNumber               := E_FunctionNumber.F_10_001_0202_01_0;
fbF_10_001_0201_01_0.ConfigFunction.NumberOfZones                     := 1;

fbF_10_001_0201_01_0.ConfigFunction.Zone[1].ZoneName                  := '10-001-0201-01-1';
fbF_10_001_0201_01_0.ConfigFunction.Zone[1].EnableMFC                 := TRUE;
fbF_10_001_0201_01_0.ConfigFunction.Zone[1].EnableLatchOccupiedState  := TRUE;
fbF_10_001_0201_01_0.ConfigFunction.Zone[1].Length[1]                 := 1200;

fbF_10_001_0201_01_0.Config.TimeoutValueLift							:= T#10S;
fbF_10_001_0201_01_0.Config.HomePosFree                               := E_Positions_LowLiftControl.DOWN;
fbF_10_001_0201_01_0.Config.HomePosOccupied                           := E_Positions_LowLiftControl.DOWN;

// Register function
FunctionRegistry[F_10_001_0201_01_0].Enable                           := TRUE; (* Function will be called *)
FunctionRegistry[F_10_001_0201_01_0].eFunctionNumber                  := fbF_10_001_0201_01_0.ConfigFunction.eFunctionNumber; // Registration number


(****************************** 10-001-0202-00-0 ************************************)
(*************************** ProBoxElement with one Motor *******************************)
// Configuration element 
fbEL_10_001_0202_00_0.ConfigElement.ElementName                     := '10-001-0202-00-0'; // Element name 
fbEL_10_001_0202_00_0.ConfigElement.eElementNumber                  := E_10_001_0202_00_0; // Number of the element 
fbEL_10_001_0202_00_0.ConfigElement.eSlaveElementNumber_34          := E_ElementNumber.E_BEGIN_ELEMENT; // Link from Master to slave element
fbEL_10_001_0202_00_0.ConfigElement.eElementType                    := E_ElementType.NO_TYPE; // No specific type

// Register element 
ElementRegistry[E_10_001_0202_00_0].Enable                          := TRUE; // Object is called
ElementRegistry[E_10_001_0202_00_0].eElementNumber                  := fbEL_10_001_0202_00_0.ConfigElement.eElementNumber; 

(****************************** 10-001-0202-01-0 ************************************)
(************************** ProBox Straight Transport *******************************)
// Configuration function
fbF_10_001_0202_01_0.ConfigFunction.FunctionName                       := '10-001-0202-01-0'; // Function name
fbF_10_001_0202_01_0.ConfigFunction.eFunctionNumber                    := F_10_001_0202_01_0; // Number of the function
fbF_10_001_0202_01_0.ConfigFunction.eElementLink                       := E_ElementNumber.E_10_001_0202_00_0;
fbF_10_001_0202_01_0.ConfigFunction.FunctionLink.eFunctionNumber       := E_FunctionNumber.F_BEGIN_FUNCTION;
fbF_10_001_0202_01_0.ConfigFunction.FunctionLink.ZoneNumber            := 0;
fbF_10_001_0202_01_0.ConfigFunction.eAdjacentFunctionNumberSide[1]     := E_FunctionNumber.F_10_001_0201_01_0;
fbF_10_001_0202_01_0.ConfigFunction.eAdjacentFunctionNumberSide[2]     := E_FunctionNumber.F_10_001_0203_01_0;
fbF_10_001_0202_01_0.ConfigFunction.ePrevFunctionNumber                := E_FunctionNumber.F_10_001_0201_01_0;
fbF_10_001_0202_01_0.ConfigFunction.eNextFunctionNumber                := E_FunctionNumber.F_10_001_0203_01_0;
fbF_10_001_0202_01_0.ConfigFunction.NumberOfZones                      := 1;
//Config zone 1
fbF_10_001_0202_01_0.ConfigFunction.Zone[1].ZoneName                   := '10-001-0202-01-1';
fbF_10_001_0202_01_0.ConfigFunction.Zone[1].EnableMFC                  := TRUE;
fbF_10_001_0202_01_0.ConfigFunction.Zone[1].EnableSimultaneousTransport:= FALSE; //Disable Simultaneous transport for multi zone functions
fbF_10_001_0202_01_0.ConfigFunction.Zone[1].EnableLatchOccupiedState   := TRUE;
fbF_10_001_0202_01_0.ConfigFunction.Zone[1].Length[1]                  := INT_TO_UINT(1600 / fbF_10_001_0202_01_0.ConfigFunction.NumberOfZones);	//Zone length (ie element length / number of zones)

// Register function
FunctionRegistry[F_10_001_0202_01_0].Enable                            := TRUE; (* Function will be called *)
FunctionRegistry[F_10_001_0202_01_0].eFunctionNumber                   := fbF_10_001_0202_01_0.ConfigFunction.eFunctionNumber; // Registration number


(****************************** 10-001-0203-00-0 ************************************)
(*************************** ProBoxElement with one Motor *******************************)
// Configuration element 
fbEL_10_001_0203_00_0.ConfigElement.ElementName                     := '10-001-0203-00-0'; // Element name 
fbEL_10_001_0203_00_0.ConfigElement.eElementNumber                  := E_10_001_0203_00_0; // Number of the element 
fbEL_10_001_0203_00_0.ConfigElement.eSlaveElementNumber_34          := E_ElementNumber.E_BEGIN_ELEMENT; // Link from Master to slave element
fbEL_10_001_0203_00_0.ConfigElement.eElementType                    := E_ElementType.NO_TYPE; // No specific type

// Register element 
ElementRegistry[E_10_001_0203_00_0].Enable                          := TRUE; // Object is called
ElementRegistry[E_10_001_0203_00_0].eElementNumber                  := fbEL_10_001_0203_00_0.ConfigElement.eElementNumber; 

(****************************** 10-001-0203-01-0 ************************************)
(************************** ProBox Straight Transport *******************************)
// Configuration function
fbF_10_001_0203_01_0.ConfigFunction.FunctionName                       := '10-001-0203-01-0'; // Function name
fbF_10_001_0203_01_0.ConfigFunction.eFunctionNumber                    := F_10_001_0203_01_0; // Number of the function
fbF_10_001_0203_01_0.ConfigFunction.eElementLink                       := E_ElementNumber.E_10_001_0203_00_0;
fbF_10_001_0203_01_0.ConfigFunction.FunctionLink.eFunctionNumber       := E_FunctionNumber.F_BEGIN_FUNCTION;
fbF_10_001_0203_01_0.ConfigFunction.FunctionLink.ZoneNumber            := 0;
fbF_10_001_0203_01_0.ConfigFunction.eAdjacentFunctionNumberSide[1]     := E_FunctionNumber.F_10_001_0202_01_0;
fbF_10_001_0203_01_0.ConfigFunction.eAdjacentFunctionNumberSide[2]     := E_FunctionNumber.F_10_001_0204_01_0;
fbF_10_001_0203_01_0.ConfigFunction.ePrevFunctionNumber                := E_FunctionNumber.F_10_001_0202_01_0;
fbF_10_001_0203_01_0.ConfigFunction.eNextFunctionNumber                := E_FunctionNumber.F_BEGIN_FUNCTION;
fbF_10_001_0203_01_0.ConfigFunction.NumberOfZones                      := 1;
//Config zone 1
fbF_10_001_0203_01_0.ConfigFunction.Zone[1].ZoneName                   := '10-001-0203-01-1';
fbF_10_001_0203_01_0.ConfigFunction.Zone[1].EnableMFC                  := TRUE;
fbF_10_001_0203_01_0.ConfigFunction.Zone[1].EnableSimultaneousTransport:= FALSE; //Disable Simultaneous transport for multi zone functions
fbF_10_001_0203_01_0.ConfigFunction.Zone[1].EnableLatchOccupiedState   := TRUE;
fbF_10_001_0203_01_0.ConfigFunction.Zone[1].Length[1]                  := INT_TO_UINT(1800 / fbF_10_001_0203_01_0.ConfigFunction.NumberOfZones);	//Zone length (ie element length / number of zones)

// Register function
FunctionRegistry[F_10_001_0203_01_0].Enable                            := TRUE; (* Function will be called *)
FunctionRegistry[F_10_001_0203_01_0].eFunctionNumber                   := fbF_10_001_0203_01_0.ConfigFunction.eFunctionNumber; // Registration number



(****************************** 10-001-0203-02-0 ************************************)
(***************************** Sick Profile Gauge ****************************)
// Configuration Profile check function
fbF_10_001_0203_02_0.ConfigFunction.FunctionName                       := '10-001-0203-02-0'; (* Function name *)
fbF_10_001_0203_02_0.ConfigFunction.eFunctionNumber                    := F_10_001_0203_02_0; (* Number of the function *)
fbF_10_001_0203_02_0.ConfigFunction.eFunctionType                      := E_FunctionType.NO_TYPE;
fbF_10_001_0203_02_0.ConfigFunction.eElementLink                       := E_ElementNumber.E_10_001_0203_00_0; 
fbF_10_001_0203_02_0.ConfigFunction.FunctionLink.eFunctionNumber       := E_FunctionNumber.F_10_001_0203_01_0;	//Addon link to function, this is auto generated, an may need to be changed.
fbF_10_001_0203_02_0.ConfigFunction.FunctionLink.ZoneNumber            := 1;		

fbF_10_001_0203_02_0.Config.ReportRealMeasureFront						:= TRUE;
fbF_10_001_0203_02_0.Config.ReportRealMeasureHeight					:= TRUE;
fbF_10_001_0203_02_0.Config.ReportRealMeasureLeft						:= TRUE;
fbF_10_001_0203_02_0.Config.ReportRealMeasureRear						:= TRUE;
fbF_10_001_0203_02_0.Config.ReportRealMeasureRight						:= TRUE;

fbF_10_001_0203_02_0.Config.EnableExternalTrigger 						:= FALSE;
fbF_10_001_0203_02_0.Config.DoubleHeightLightGrids 					:= FALSE;
fbF_10_001_0203_02_0.Config.BeamSpacing_HeightLower					:= 20;
fbF_10_001_0203_02_0.Config.BeamSpacing_HeightUpper					:= 20;
fbF_10_001_0203_02_0.Config.BeamSpacing_WidthLeft						:= 5;
fbF_10_001_0203_02_0.Config.BeamSpacing_WidthRight						:= 5;
fbF_10_001_0203_02_0.Config.BeamSpacing_Length							:= 5;
fbF_10_001_0203_02_0.Config.ReportValue_Measurement_Error_Left			:= 2;
fbF_10_001_0203_02_0.Config.ReportValue_Measurement_Error_Right		:= 2;
fbF_10_001_0203_02_0.Config.ReportValue_Measurement_Error_Height		:= 9;
fbF_10_001_0203_02_0.Config.ReportValue_Measurement_Error_Front		:= 2;
fbF_10_001_0203_02_0.Config.ReportValue_Measurement_Error_Rear			:= 2;
fbF_10_001_0203_02_0.Config.LightGrid_Offset_Height_Lower 				:= 100;
fbF_10_001_0203_02_0.Config.LightGrid_Offset_Height_Upper				:= 0;
fbF_10_001_0203_02_0.Config.LightGrid_Offset_Width_Left				:= 135;
fbF_10_001_0203_02_0.Config.LightGrid_Offset_Width_Right				:= 90;
fbF_10_001_0203_02_0.Config.LightGrid_Offset_Length_Front				:= 155;
fbF_10_001_0203_02_0.Config.LightGrid_Offset_Length_Rear				:= 155;
              
fbF_10_001_0203_02_0.Config.ProfileRule_Height[1].TU_Type				:= 0;
fbF_10_001_0203_02_0.Config.ProfileRule_Height[1].Minimum				:= 200;
fbF_10_001_0203_02_0.Config.ProfileRule_Height[1].Maximum				:= 1200;
fbF_10_001_0203_02_0.Config.ProfileRule_Height[1].ReportValue			:= 1;
fbF_10_001_0203_02_0.Config.ProfileRule_Height[1].Default				:= 0;
            
fbF_10_001_0203_02_0.Config.ProfileRule_OverhangLeft[1].TU_Type		:= 0;
fbF_10_001_0203_02_0.Config.ProfileRule_OverhangLeft[1].ReportValue	:= 1;
fbF_10_001_0203_02_0.Config.ProfileRule_OverhangLeft[1].Minimum		:= 0;
fbF_10_001_0203_02_0.Config.ProfileRule_OverhangLeft[1].Maximum		:= 50;
fbF_10_001_0203_02_0.Config.ProfileRule_OverhangLeft[1].Default		:= 400;
             
fbF_10_001_0203_02_0.Config.ProfileRule_OverhangRight[1].TU_Type		:= 0;
fbF_10_001_0203_02_0.Config.ProfileRule_OverhangRight[1].ReportValue 	:= 1;
fbF_10_001_0203_02_0.Config.ProfileRule_OverhangRight[1].Minimum		:= 0;
fbF_10_001_0203_02_0.Config.ProfileRule_OverhangRight[1].Maximum		:= 50;
fbF_10_001_0203_02_0.Config.ProfileRule_OverhangRight[1].Default		:= 400;
           
fbF_10_001_0203_02_0.Config.ProfileRule_OverhangFront[1].TU_Type		:= 0;
fbF_10_001_0203_02_0.Config.ProfileRule_OverhangFront[1].ReportValue	:= 1;
fbF_10_001_0203_02_0.Config.ProfileRule_OverhangFront[1].Minimum		:= 0;
fbF_10_001_0203_02_0.Config.ProfileRule_OverhangFront[1].Maximum		:= 50;
fbF_10_001_0203_02_0.Config.ProfileRule_OverhangFront[1].Default		:= 600;
            
fbF_10_001_0203_02_0.Config.ProfileRule_OverhangRear[1].TU_Type			:= 0;
fbF_10_001_0203_02_0.Config.ProfileRule_OverhangRear[1].ReportValue		:= 1;
fbF_10_001_0203_02_0.Config.ProfileRule_OverhangRear[1].Minimum			:= 0;
fbF_10_001_0203_02_0.Config.ProfileRule_OverhangRear[1].Maximum			:= 50;
fbF_10_001_0203_02_0.Config.ProfileRule_OverhangRear[1].Default			:= 600;


// Register function 
FunctionRegistry[F_10_001_0203_02_0].Enable                     		:= TRUE; (* Function will be called *)
FunctionRegistry[F_10_001_0203_02_0].eFunctionNumber 					:= fbF_10_001_0203_02_0.ConfigFunction.eFunctionNumber; // Registration number 

(****************************** 10-001-0203-03-0 ************************************)
(****************************** SICK Scanner CLV 6xx **************************************)
// Configuration function 
fbF_10_001_0203_03_0.ConfigFunction.FunctionName                     := '10-001-0203-03-0'; (* Function name *)
fbF_10_001_0203_03_0.ConfigFunction.eFunctionNumber                  := F_10_001_0203_03_0; (* Number of the function *)
fbF_10_001_0203_03_0.ConfigFunction.eFunctionType                    := E_FunctionType.NO_TYPE;
fbF_10_001_0203_03_0.ConfigFunction.eElementLink                     := E_ElementNumber.E_10_001_0203_00_0; 
fbF_10_001_0203_03_0.ConfigFunction.FunctionLink.eFunctionNumber     := E_FunctionNumber.F_10_001_0203_01_0;	//Addon link to function, this is auto generated, an may need to be changed.
fbF_10_001_0203_03_0.ConfigFunction.FunctionLink.ZoneNumber          := 1;		

fbF_10_001_0203_03_0.Config.MaxLabelLength                           := 18; // Maximum label length
fbF_10_001_0203_03_0.Config.EnableExternalTrigger					  := FALSE; 
fbF_10_001_0203_03_0.Config.AcceptedNoReadSeries					  := 5; // 0 = disabled. Number of accepted no reads before setting an error.
fbF_10_001_0203_03_0.Config.tComTimeout                              := T#5S; // Scanner heartbeat signal timeout
fbF_10_001_0203_03_0.Config.SendTTQ                                  := FALSE; // Send TTQ
fbF_10_001_0203_03_0.Config.MoveDataLabelField                       := TRUE; //Barcode written to lable field. If false, move data to TU ID
fbF_10_001_0203_03_0.Config.ConfigFilePath                           := ''; //Path to file to write to scanner during State CONFIG. Empty = not enabled

// Register function 
FunctionRegistry[F_10_001_0203_03_0].Enable                           := TRUE; (* Function will be called *)
FunctionRegistry[F_10_001_0203_03_0].eFunctionNumber                  := fbF_10_001_0203_03_0.ConfigFunction.eFunctionNumber; (* Registration number *)


(****************************** 10-001-0203-04-0 ************************************)
(******************************** TLB4 Weight ***************************************)
// Configuration function 
fbF_10_001_0203_04_0.ConfigFunction.FunctionName                     := '10-001-0203-04-0'; (* Function name *)
fbF_10_001_0203_04_0.ConfigFunction.eFunctionNumber                  := F_10_001_0203_04_0; (* Number of the function *)
fbF_10_001_0203_04_0.ConfigFunction.eFunctionType                    := E_FunctionType.NO_TYPE;
fbF_10_001_0203_04_0.ConfigFunction.eElementLink                     := E_ElementNumber.E_10_001_0203_00_0; 
fbF_10_001_0203_04_0.ConfigFunction.FunctionLink.eFunctionNumber     := E_FunctionNumber.F_10_001_0203_01_0;	//Addon link to function, this is auto generated, an may need to be changed.
fbF_10_001_0203_04_0.ConfigFunction.FunctionLink.ZoneNumber          := 1;		

fbF_10_001_0203_04_0.Config.MaxDiffFromZero							:= 30;
fbF_10_001_0203_04_0.Config.MaxWeight								:= 1000000;
fbF_10_001_0203_04_0.Config.MinWeight								:= 0;
fbF_10_001_0203_04_0.Config.WaitForStability						:= TRUE;

// Register function 
FunctionRegistry[F_10_001_0203_04_0].Enable                           := TRUE; (* Function will be called *)
FunctionRegistry[F_10_001_0203_04_0].eFunctionNumber                  := fbF_10_001_0203_04_0.ConfigFunction.eFunctionNumber; (* Registration number *)


(****************************** 10-001-0203-05-0 ************************************)
(******************************** PalletCheckAddon ***************************************)
// Configuration function 
fbF_10_001_0203_05_0.ConfigFunction.FunctionName                     := '10-001-0203-05-0'; (* Function name *)
fbF_10_001_0203_05_0.ConfigFunction.eFunctionNumber                  := F_10_001_0203_05_0; (* Number of the function *)
fbF_10_001_0203_05_0.ConfigFunction.eFunctionType                    := E_FunctionType.NO_TYPE;
fbF_10_001_0203_05_0.ConfigFunction.eElementLink                     := E_ElementNumber.E_10_001_0203_00_0; 
fbF_10_001_0203_05_0.ConfigFunction.FunctionLink.eFunctionNumber     := E_FunctionNumber.F_10_001_0203_01_0;	//Addon link to function, this is auto generated, an may need to be changed.
fbF_10_001_0203_05_0.ConfigFunction.FunctionLink.ZoneNumber          := 1;		


fbF_10_001_0203_05_0.Config.EnableExternalTrigger 						:= FALSE;


// Register function
FunctionRegistry[F_10_001_0203_05_0].Enable                           := TRUE; (* Function will be called *)
FunctionRegistry[F_10_001_0203_05_0].eFunctionNumber                  := fbF_10_001_0203_05_0.ConfigFunction.eFunctionNumber; (* Registration number *)




(****************************** 10-001-0204-00-0 ************************************)
(*************************** ProBoxElement with one Motor *******************************)
// Configuration element 
fbEL_10_001_0204_00_0.ConfigElement.ElementName                     := '10-001-0204-00-0'; // Element name 
fbEL_10_001_0204_00_0.ConfigElement.eElementNumber                  := E_10_001_0204_00_0; // Number of the element 
fbEL_10_001_0204_00_0.ConfigElement.eSlaveElementNumber_34          := E_ElementNumber.E_BEGIN_ELEMENT; // Link from Master to slave element
fbEL_10_001_0204_00_0.ConfigElement.eElementType                    := E_ElementType.NO_TYPE; // No specific type

// Register element 
ElementRegistry[E_10_001_0204_00_0].Enable                          := TRUE; // Object is called
ElementRegistry[E_10_001_0204_00_0].eElementNumber                  := fbEL_10_001_0204_00_0.ConfigElement.eElementNumber; 

(****************************** 10-001-0204-01-0 ************************************)
(******************************** TurnTable with one drive *************************************)
// Configuration function
fbF_10_001_0204_01_0.ConfigFunction.FunctionName                      := '10-001-0204-01-0'; // Function name
fbF_10_001_0204_01_0.ConfigFunction.eFunctionNumber                   := F_10_001_0204_01_0; // Number of the function
fbF_10_001_0204_01_0.ConfigFunction.eElementLink                      := E_ElementNumber.E_10_001_0204_00_0;
fbF_10_001_0204_01_0.ConfigFunction.FunctionLink.eFunctionNumber      := E_FunctionNumber.F_BEGIN_FUNCTION;
fbF_10_001_0204_01_0.ConfigFunction.FunctionLink.ZoneNumber           := 0;
fbF_10_001_0204_01_0.ConfigFunction.eAdjacentFunctionNumberSide[1]    := E_FunctionNumber.F_10_001_0203_01_0;
fbF_10_001_0204_01_0.ConfigFunction.eAdjacentFunctionNumberSide[2]    := E_FunctionNumber.F_10_001_0233_01_0;
fbF_10_001_0204_01_0.ConfigFunction.eAdjacentFunctionNumberSide[4]    := E_FunctionNumber.F_10_002_0206_01_0;
fbF_10_001_0204_01_0.ConfigFunction.ePrevFunctionNumber               := E_FunctionNumber.F_10_001_0203_01_0;
fbF_10_001_0204_01_0.ConfigFunction.eNextFunctionNumber               := E_FunctionNumber.F_BEGIN_FUNCTION;
fbF_10_001_0204_01_0.ConfigFunction.FlowDirectionREV                  := FALSE;
fbF_10_001_0204_01_0.ConfigFunction.NumberOfZones                     := 1;

fbF_10_001_0204_01_0.ConfigFunction.Zone[1].ZoneName                  := '10-001-0204-01-1';
fbF_10_001_0204_01_0.ConfigFunction.Zone[1].EnableMFC                 := TRUE;
fbF_10_001_0204_01_0.ConfigFunction.Zone[1].EnableLatchOccupiedState  := TRUE;
fbF_10_001_0204_01_0.ConfigFunction.Zone[1].Length[1]                 := 1000;

fbF_10_001_0204_01_0.Config.TurnHomePosFree                           := E_Positions_TurnControl.MIDDLE;
fbF_10_001_0204_01_0.Config.TurnHomePosOccupied                       := E_Positions_TurnControl.CW;
fbF_10_001_0204_01_0.Config.TurnTimeoutValue                          := T#15S;

// Register function
FunctionRegistry[F_10_001_0204_01_0].Enable                           := TRUE; (* Function will be called *)
FunctionRegistry[F_10_001_0204_01_0].eFunctionNumber                  := fbF_10_001_0204_01_0.ConfigFunction.eFunctionNumber; // Registration number


(****************************** 10-001-0205-00-0 ************************************)
(*************************** ProBoxElement with one Motor *******************************)
// Configuration element 
fbEL_10_001_0205_00_0.ConfigElement.ElementName                     := '10-001-0205-00-0'; // Element name 
fbEL_10_001_0205_00_0.ConfigElement.eElementNumber                  := E_10_001_0205_00_0; // Number of the element 
fbEL_10_001_0205_00_0.ConfigElement.eSlaveElementNumber_34          := E_ElementNumber.E_BEGIN_ELEMENT; // Link from Master to slave element
fbEL_10_001_0205_00_0.ConfigElement.eElementType                    := E_ElementType.NO_TYPE; // No specific type

// Register element 
ElementRegistry[E_10_001_0205_00_0].Enable                          := TRUE; // Object is called
ElementRegistry[E_10_001_0205_00_0].eElementNumber                  := fbEL_10_001_0205_00_0.ConfigElement.eElementNumber; 

(****************************** 10-001-0207-00-0 ************************************)
(*************************** ProBoxElement with one Motor *******************************)
// Configuration element 
fbEL_10_001_0207_00_0.ConfigElement.ElementName                     := '10-001-0207-00-0'; // Element name 
fbEL_10_001_0207_00_0.ConfigElement.eElementNumber                  := E_10_001_0207_00_0; // Number of the element 
fbEL_10_001_0207_00_0.ConfigElement.eSlaveElementNumber_34          := E_ElementNumber.E_BEGIN_ELEMENT; // Link from Master to slave element
fbEL_10_001_0207_00_0.ConfigElement.eElementType                    := E_ElementType.NO_TYPE; // No specific type

// Register element 
ElementRegistry[E_10_001_0207_00_0].Enable                          := TRUE; // Object is called
ElementRegistry[E_10_001_0207_00_0].eElementNumber                  := fbEL_10_001_0207_00_0.ConfigElement.eElementNumber; 

(****************************** 10-001-0207-01-0 ************************************)
(************************** ProBox Straight Transport *******************************)
// Configuration function
fbF_10_001_0207_01_0.ConfigFunction.FunctionName                       := '10-001-0207-01-0'; // Function name
fbF_10_001_0207_01_0.ConfigFunction.eFunctionNumber                    := F_10_001_0207_01_0; // Number of the function
fbF_10_001_0207_01_0.ConfigFunction.eElementLink                       := E_ElementNumber.E_10_001_0207_00_0;
fbF_10_001_0207_01_0.ConfigFunction.FunctionLink.eFunctionNumber       := E_FunctionNumber.F_BEGIN_FUNCTION;
fbF_10_001_0207_01_0.ConfigFunction.FunctionLink.ZoneNumber            := 0;
fbF_10_001_0207_01_0.ConfigFunction.eAdjacentFunctionNumberSide[1]     := E_FunctionNumber.F_BEGIN_FUNCTION;
fbF_10_001_0207_01_0.ConfigFunction.eAdjacentFunctionNumberSide[2]     := E_FunctionNumber.F_BEGIN_FUNCTION;
fbF_10_001_0207_01_0.ConfigFunction.ePrevFunctionNumber                := E_FunctionNumber.F_BEGIN_FUNCTION;
fbF_10_001_0207_01_0.ConfigFunction.eNextFunctionNumber                := E_FunctionNumber.F_BEGIN_FUNCTION;
fbF_10_001_0207_01_0.ConfigFunction.NumberOfZones                      := 1;
//Config zone 1
fbF_10_001_0207_01_0.ConfigFunction.Zone[1].ZoneName                   := '10-001-0207-01-1';
fbF_10_001_0207_01_0.ConfigFunction.Zone[1].EnableMFC                  := TRUE;
fbF_10_001_0207_01_0.ConfigFunction.Zone[1].EnableSimultaneousTransport:= FALSE; //Disable Simultaneous transport for multi zone functions
fbF_10_001_0207_01_0.ConfigFunction.Zone[1].EnableLatchOccupiedState   := TRUE;
fbF_10_001_0207_01_0.ConfigFunction.Zone[1].Length[1]                  := INT_TO_UINT(1500 / fbF_10_001_0207_01_0.ConfigFunction.NumberOfZones);	//Zone length (ie element length / number of zones)

// Register function
FunctionRegistry[F_10_001_0207_01_0].Enable                            := TRUE; (* Function will be called *)
FunctionRegistry[F_10_001_0207_01_0].eFunctionNumber                   := fbF_10_001_0207_01_0.ConfigFunction.eFunctionNumber; // Registration number


(****************************** 10-001-0207-02-0 ************************************)
(****************************** PalletMagazine Addon *************************************)
// Configuration function 
fbF_10_001_0207_02_0.ConfigFunction.FunctionName					:= '10-001-0207-02-0'; (* Function name *)
fbF_10_001_0207_02_0.ConfigFunction.eFunctionNumber				:= F_10_001_0207_02_0; (* Number of the function *)
fbF_10_001_0207_02_0.ConfigFunction.eFunctionType					:= E_FunctionType.NO_TYPE;
fbF_10_001_0207_02_0.ConfigFunction.eElementLink					:= E_ElementNumber.E_10_001_0207_00_0; 
fbF_10_001_0207_02_0.ConfigFunction.FunctionLink.eFunctionNumber	:= E_FunctionNumber.F_10_001_0207_01_0;	//Addon link to function, this is auto generated, an may need to be changed.
fbF_10_001_0207_02_0.ConfigFunction.FunctionLink.ZoneNumber		:= 1;		

fbF_10_001_0207_02_0.Config.TimeoutValueLift						:= T#20S; //Timeout when moving lift
fbF_10_001_0207_02_0.Config.TimeoutValueSeq						:= T#2M;  //Timeout for complete sequence
fbF_10_001_0207_02_0.Config.IdleStacking							:= FALSE; //Lift pallet up to optimze stacking

// Register function 
FunctionRegistry[F_10_001_0207_02_0].Enable                           := TRUE; (* Function will be called *)
FunctionRegistry[F_10_001_0207_02_0].eFunctionNumber                  := fbF_10_001_0207_02_0.ConfigFunction.eFunctionNumber; (* Registration number *)

(****************************** 10-001-0208-00-0 ************************************)
(*************************** ProBoxElement with one Motor *******************************)
// Configuration element 
fbEL_10_001_0208_00_0.ConfigElement.ElementName                     := '10-001-0208-00-0'; // Element name 
fbEL_10_001_0208_00_0.ConfigElement.eElementNumber                  := E_10_001_0208_00_0; // Number of the element 
fbEL_10_001_0208_00_0.ConfigElement.eSlaveElementNumber_34          := E_ElementNumber.E_BEGIN_ELEMENT; // Link from Master to slave element
fbEL_10_001_0208_00_0.ConfigElement.eElementType                    := E_ElementType.NO_TYPE; // No specific type

// Register element 
ElementRegistry[E_10_001_0208_00_0].Enable                          := TRUE; // Object is called
ElementRegistry[E_10_001_0208_00_0].eElementNumber                  := fbEL_10_001_0208_00_0.ConfigElement.eElementNumber; 

(****************************** 10-001-0208-01-0 ************************************)
(************************** ProBox Straight Transport *******************************)
// Configuration function
fbF_10_001_0208_01_0.ConfigFunction.FunctionName                       := '10-001-0208-01-0'; // Function name
fbF_10_001_0208_01_0.ConfigFunction.eFunctionNumber                    := F_10_001_0208_01_0; // Number of the function
fbF_10_001_0208_01_0.ConfigFunction.eElementLink                       := E_ElementNumber.E_10_001_0208_00_0;
fbF_10_001_0208_01_0.ConfigFunction.FunctionLink.eFunctionNumber       := E_FunctionNumber.F_BEGIN_FUNCTION;
fbF_10_001_0208_01_0.ConfigFunction.FunctionLink.ZoneNumber            := 0;
fbF_10_001_0208_01_0.ConfigFunction.eAdjacentFunctionNumberSide[1]     := E_FunctionNumber.F_10_002_0206_01_0;
fbF_10_001_0208_01_0.ConfigFunction.eAdjacentFunctionNumberSide[2]     := E_FunctionNumber.F_10_001_0209_01_0;
fbF_10_001_0208_01_0.ConfigFunction.ePrevFunctionNumber                := E_FunctionNumber.F_10_002_0206_01_0;
fbF_10_001_0208_01_0.ConfigFunction.eNextFunctionNumber                := E_FunctionNumber.F_10_001_0209_01_0;
fbF_10_001_0208_01_0.ConfigFunction.NumberOfZones                      := 1;
//Config zone 1
fbF_10_001_0208_01_0.ConfigFunction.Zone[1].ZoneName                   := '10-001-0208-01-1';
fbF_10_001_0208_01_0.ConfigFunction.Zone[1].EnableMFC                  := TRUE;
fbF_10_001_0208_01_0.ConfigFunction.Zone[1].EnableSimultaneousTransport:= FALSE; //Disable Simultaneous transport for multi zone functions
fbF_10_001_0208_01_0.ConfigFunction.Zone[1].EnableLatchOccupiedState   := TRUE;
fbF_10_001_0208_01_0.ConfigFunction.Zone[1].Length[1]                  := INT_TO_UINT(1800 / fbF_10_001_0208_01_0.ConfigFunction.NumberOfZones);	//Zone length (ie element length / number of zones)

// Register function
FunctionRegistry[F_10_001_0208_01_0].Enable                            := TRUE; (* Function will be called *)
FunctionRegistry[F_10_001_0208_01_0].eFunctionNumber                   := fbF_10_001_0208_01_0.ConfigFunction.eFunctionNumber; // Registration number


(****************************** 10-001-0209-00-0 ************************************)
(*************************** ProBoxElement with one Motor *******************************)
// Configuration element 
fbEL_10_001_0209_00_0.ConfigElement.ElementName                     := '10-001-0209-00-0'; // Element name 
fbEL_10_001_0209_00_0.ConfigElement.eElementNumber                  := E_10_001_0209_00_0; // Number of the element 
fbEL_10_001_0209_00_0.ConfigElement.eSlaveElementNumber_34          := E_ElementNumber.E_10_001_0214_00_0; // Link from Master to slave element
fbEL_10_001_0209_00_0.ConfigElement.eElementType                    := E_ElementType.NO_TYPE; // No specific type

// Register element 
ElementRegistry[E_10_001_0209_00_0].Enable                          := TRUE; // Object is called
ElementRegistry[E_10_001_0209_00_0].eElementNumber                  := fbEL_10_001_0209_00_0.ConfigElement.eElementNumber; 

(****************************** 10-001-0209-01-0 ************************************)
(******************************** Transfer Unit *************************************)
// Configuration function
fbF_10_001_0209_01_0.ConfigFunction.FunctionName                    := '10-001-0209-01-0'; // Function name
fbF_10_001_0209_01_0.ConfigFunction.eFunctionNumber                 := F_10_001_0209_01_0; // Number of the function
fbF_10_001_0209_01_0.ConfigFunction.eElementLink                    := E_ElementNumber.E_10_001_0209_00_0;
fbF_10_001_0209_01_0.ConfigFunction.FunctionLink.eFunctionNumber    := E_FunctionNumber.F_BEGIN_FUNCTION;
fbF_10_001_0209_01_0.ConfigFunction.FunctionLink.ZoneNumber         := 0;
fbF_10_001_0209_01_0.ConfigFunction.eAdjacentFunctionNumberSide[1]  := E_FunctionNumber.F_10_001_0208_01_0;
fbF_10_001_0209_01_0.ConfigFunction.eAdjacentFunctionNumberSide[2]  := E_FunctionNumber.F_10_001_0211_01_0;
fbF_10_001_0209_01_0.ConfigFunction.eAdjacentFunctionNumberSide[3]  := E_FunctionNumber.F_10_001_0227_01_0;
fbF_10_001_0209_01_0.ConfigFunction.eAdjacentFunctionNumberSide[4]  := E_FunctionNumber.F_10_001_0214_01_0;
fbF_10_001_0209_01_0.ConfigFunction.ePrevFunctionNumber             := E_FunctionNumber.F_BEGIN_FUNCTION;
fbF_10_001_0209_01_0.ConfigFunction.eNextFunctionNumber             := E_FunctionNumber.F_BEGIN_FUNCTION;
fbF_10_001_0209_01_0.ConfigFunction.FlowDirectionREV                := FALSE;
fbF_10_001_0209_01_0.ConfigFunction.NumberOfZones                   := 1;

fbF_10_001_0209_01_0.ConfigFunction.Zone[1].ZoneName                := '10-001-0209-01-1';
fbF_10_001_0209_01_0.ConfigFunction.Zone[1].EnableMFC                 := TRUE;
fbF_10_001_0209_01_0.ConfigFunction.Zone[1].EnableLatchOccupiedState  := TRUE;
fbF_10_001_0209_01_0.ConfigFunction.Zone[1].Length[1]               := 1000;

fbF_10_001_0209_01_0.Config.TimeoutValueLift                        := T#15S; // Timeout value for lifting
fbF_10_001_0209_01_0.Config.HomePosFree                             := E_Positions_LiftControl.UP; // Homeposition lift when zone free, UNDIFINED=> No home position is set, and lift stays where it is.
fbF_10_001_0209_01_0.Config.HomePosOccupied                         := E_Positions_LiftControl.DOWN; // Homeposition lift when zone occupied, UNDIFINED=> No home position is set, and lift stays where it is.
fbF_10_001_0209_01_0.Config.LiftType                                := E_LiftType.E_LiftChain; // Configured lifting type, Roller or Chain
fbF_10_001_0209_01_0.Config.SingleTUMode							 := E_SingleTuMode.SingleTuMode; // Transfer unit and slave element's extended functions only allow one TU at a time. Change to optimize the transfer unit.

// Register function                                                     
FunctionRegistry[F_10_001_0209_01_0].Enable                         := TRUE; (* Function will be called *)
FunctionRegistry[F_10_001_0209_01_0].eFunctionNumber                := fbF_10_001_0209_01_0.ConfigFunction.eFunctionNumber; // Registration number


(****************************** 10-001-0211-00-0 ************************************)
(*************************** ProBoxElement with one Motor *******************************)
// Configuration element 
fbEL_10_001_0211_00_0.ConfigElement.ElementName                     := '10-001-0211-00-0'; // Element name 
fbEL_10_001_0211_00_0.ConfigElement.eElementNumber                  := E_10_001_0211_00_0; // Number of the element 
fbEL_10_001_0211_00_0.ConfigElement.eSlaveElementNumber_34          := E_ElementNumber.E_BEGIN_ELEMENT; // Link from Master to slave element
fbEL_10_001_0211_00_0.ConfigElement.eElementType                    := E_ElementType.NO_TYPE; // No specific type

// Register element 
ElementRegistry[E_10_001_0211_00_0].Enable                          := TRUE; // Object is called
ElementRegistry[E_10_001_0211_00_0].eElementNumber                  := fbEL_10_001_0211_00_0.ConfigElement.eElementNumber; 

(****************************** 10-001-0211-01-0 ************************************)
(************************** ProBox Straight Transport *******************************)
// Configuration function
fbF_10_001_0211_01_0.ConfigFunction.FunctionName                       := '10-001-0211-01-0'; // Function name
fbF_10_001_0211_01_0.ConfigFunction.eFunctionNumber                    := F_10_001_0211_01_0; // Number of the function
fbF_10_001_0211_01_0.ConfigFunction.eElementLink                       := E_ElementNumber.E_10_001_0211_00_0;
fbF_10_001_0211_01_0.ConfigFunction.FunctionLink.eFunctionNumber       := E_FunctionNumber.F_BEGIN_FUNCTION;
fbF_10_001_0211_01_0.ConfigFunction.FunctionLink.ZoneNumber            := 0;
fbF_10_001_0211_01_0.ConfigFunction.eAdjacentFunctionNumberSide[1]     := E_FunctionNumber.F_10_001_0209_01_0;
fbF_10_001_0211_01_0.ConfigFunction.eAdjacentFunctionNumberSide[2]     := E_FunctionNumber.F_10_001_0212_01_0;
fbF_10_001_0211_01_0.ConfigFunction.ePrevFunctionNumber                := E_FunctionNumber.F_10_001_0209_01_0;
fbF_10_001_0211_01_0.ConfigFunction.eNextFunctionNumber                := E_FunctionNumber.F_10_001_0212_01_0;
fbF_10_001_0211_01_0.ConfigFunction.NumberOfZones                      := 1;
//Config zone 1
fbF_10_001_0211_01_0.ConfigFunction.Zone[1].ZoneName                   := '10-001-0211-01-1';
fbF_10_001_0211_01_0.ConfigFunction.Zone[1].EnableMFC                  := TRUE;
fbF_10_001_0211_01_0.ConfigFunction.Zone[1].EnableSimultaneousTransport:= FALSE; //Disable Simultaneous transport for multi zone functions
fbF_10_001_0211_01_0.ConfigFunction.Zone[1].EnableLatchOccupiedState   := TRUE;
fbF_10_001_0211_01_0.ConfigFunction.Zone[1].Length[1]                  := INT_TO_UINT(1400 / fbF_10_001_0211_01_0.ConfigFunction.NumberOfZones);	//Zone length (ie element length / number of zones)

// Register function
FunctionRegistry[F_10_001_0211_01_0].Enable                            := TRUE; (* Function will be called *)
FunctionRegistry[F_10_001_0211_01_0].eFunctionNumber                   := fbF_10_001_0211_01_0.ConfigFunction.eFunctionNumber; // Registration number


(****************************** 10-001-0212-00-0 ************************************)
(*************************** ProBoxElement with one Motor *******************************)
// Configuration element 
fbEL_10_001_0212_00_0.ConfigElement.ElementName                     := '10-001-0212-00-0'; // Element name 
fbEL_10_001_0212_00_0.ConfigElement.eElementNumber                  := E_10_001_0212_00_0; // Number of the element 
fbEL_10_001_0212_00_0.ConfigElement.eSlaveElementNumber_34          := E_ElementNumber.E_10_001_0217_00_0; // Link from Master to slave element
fbEL_10_001_0212_00_0.ConfigElement.eElementType                    := E_ElementType.NO_TYPE; // No specific type

// Register element 
ElementRegistry[E_10_001_0212_00_0].Enable                          := TRUE; // Object is called
ElementRegistry[E_10_001_0212_00_0].eElementNumber                  := fbEL_10_001_0212_00_0.ConfigElement.eElementNumber; 

(****************************** 10-001-0212-01-0 ************************************)
(******************************** Transfer Unit *************************************)
// Configuration function
fbF_10_001_0212_01_0.ConfigFunction.FunctionName                    := '10-001-0212-01-0'; // Function name
fbF_10_001_0212_01_0.ConfigFunction.eFunctionNumber                 := F_10_001_0212_01_0; // Number of the function
fbF_10_001_0212_01_0.ConfigFunction.eElementLink                    := E_ElementNumber.E_10_001_0212_00_0;
fbF_10_001_0212_01_0.ConfigFunction.FunctionLink.eFunctionNumber    := E_FunctionNumber.F_BEGIN_FUNCTION;
fbF_10_001_0212_01_0.ConfigFunction.FunctionLink.ZoneNumber         := 0;
fbF_10_001_0212_01_0.ConfigFunction.eAdjacentFunctionNumberSide[1]  := E_FunctionNumber.F_10_001_0211_01_0;
fbF_10_001_0212_01_0.ConfigFunction.eAdjacentFunctionNumberSide[2]  := E_FunctionNumber.F_10_001_0213_01_0;
fbF_10_001_0212_01_0.ConfigFunction.eAdjacentFunctionNumberSide[3]  := E_FunctionNumber.F_10_001_0217_01_0;
fbF_10_001_0212_01_0.ConfigFunction.eAdjacentFunctionNumberSide[4]  := E_FunctionNumber.F_10_001_0218_01_0;
fbF_10_001_0212_01_0.ConfigFunction.ePrevFunctionNumber             := E_FunctionNumber.F_BEGIN_FUNCTION;
fbF_10_001_0212_01_0.ConfigFunction.eNextFunctionNumber             := E_FunctionNumber.F_BEGIN_FUNCTION;
fbF_10_001_0212_01_0.ConfigFunction.FlowDirectionREV                := FALSE;
fbF_10_001_0212_01_0.ConfigFunction.NumberOfZones                   := 1;

fbF_10_001_0212_01_0.ConfigFunction.Zone[1].ZoneName                := '10-001-0212-01-1';
fbF_10_001_0212_01_0.ConfigFunction.Zone[1].EnableMFC                 := TRUE;
fbF_10_001_0212_01_0.ConfigFunction.Zone[1].EnableLatchOccupiedState  := TRUE;
fbF_10_001_0212_01_0.ConfigFunction.Zone[1].Length[1]               := 1000;

fbF_10_001_0212_01_0.Config.TimeoutValueLift                        := T#15S; // Timeout value for lifting
fbF_10_001_0212_01_0.Config.HomePosFree                             := E_Positions_LiftControl.UNDIFINED; // Homeposition lift when zone free, UNDIFINED=> No home position is set, and lift stays where it is.
fbF_10_001_0212_01_0.Config.HomePosOccupied                         := E_Positions_LiftControl.UNDIFINED; // Homeposition lift when zone occupied, UNDIFINED=> No home position is set, and lift stays where it is.
fbF_10_001_0212_01_0.Config.LiftType                                := E_LiftType.E_LiftChain; // Configured lifting type, Roller or Chain
fbF_10_001_0212_01_0.Config.SingleTUMode							 := E_SingleTuMode.SingleTuMode; // Transfer unit and slave element's extended functions only allow one TU at a time. Change to optimize the transfer unit.

// Register function                                                     
FunctionRegistry[F_10_001_0212_01_0].Enable                         := TRUE; (* Function will be called *)
FunctionRegistry[F_10_001_0212_01_0].eFunctionNumber                := fbF_10_001_0212_01_0.ConfigFunction.eFunctionNumber; // Registration number


(****************************** 10-001-0213-00-0 ************************************)
(*************************** ProBoxElement with one Motor *******************************)
// Configuration element 
fbEL_10_001_0213_00_0.ConfigElement.ElementName                     := '10-001-0213-00-0'; // Element name 
fbEL_10_001_0213_00_0.ConfigElement.eElementNumber                  := E_10_001_0213_00_0; // Number of the element 
fbEL_10_001_0213_00_0.ConfigElement.eSlaveElementNumber_34          := E_ElementNumber.E_BEGIN_ELEMENT; // Link from Master to slave element
fbEL_10_001_0213_00_0.ConfigElement.eElementType                    := E_ElementType.NO_TYPE; // No specific type

// Register element 
ElementRegistry[E_10_001_0213_00_0].Enable                          := TRUE; // Object is called
ElementRegistry[E_10_001_0213_00_0].eElementNumber                  := fbEL_10_001_0213_00_0.ConfigElement.eElementNumber; 

(****************************** 10-001-0213-01-0 ************************************)
(************************** ProBox Straight Transport *******************************)
// Configuration function
fbF_10_001_0213_01_0.ConfigFunction.FunctionName                       := '10-001-0213-01-0'; // Function name
fbF_10_001_0213_01_0.ConfigFunction.eFunctionNumber                    := F_10_001_0213_01_0; // Number of the function
fbF_10_001_0213_01_0.ConfigFunction.eElementLink                       := E_ElementNumber.E_10_001_0213_00_0;
fbF_10_001_0213_01_0.ConfigFunction.FunctionLink.eFunctionNumber       := E_FunctionNumber.F_BEGIN_FUNCTION;
fbF_10_001_0213_01_0.ConfigFunction.FunctionLink.ZoneNumber            := 0;
fbF_10_001_0213_01_0.ConfigFunction.eAdjacentFunctionNumberSide[1]     := E_FunctionNumber.F_10_001_0212_01_0;
fbF_10_001_0213_01_0.ConfigFunction.eAdjacentFunctionNumberSide[2]     := E_FunctionNumber.F_BEGIN_FUNCTION;
fbF_10_001_0213_01_0.ConfigFunction.ePrevFunctionNumber                := E_FunctionNumber.F_10_001_0212_01_0;
fbF_10_001_0213_01_0.ConfigFunction.eNextFunctionNumber                := E_FunctionNumber.F_BEGIN_FUNCTION;
fbF_10_001_0213_01_0.ConfigFunction.NumberOfZones                      := 1;
//Config zone 1
fbF_10_001_0213_01_0.ConfigFunction.Zone[1].ZoneName                   := '10-001-0213-01-1';
fbF_10_001_0213_01_0.ConfigFunction.Zone[1].EnableMFC                  := TRUE;
fbF_10_001_0213_01_0.ConfigFunction.Zone[1].EnableSimultaneousTransport:= FALSE; //Disable Simultaneous transport for multi zone functions
fbF_10_001_0213_01_0.ConfigFunction.Zone[1].EnableLatchOccupiedState   := TRUE;
fbF_10_001_0213_01_0.ConfigFunction.Zone[1].Length[1]                  := INT_TO_UINT(1500 / fbF_10_001_0213_01_0.ConfigFunction.NumberOfZones);	//Zone length (ie element length / number of zones)

// Register function
FunctionRegistry[F_10_001_0213_01_0].Enable                            := TRUE; (* Function will be called *)
FunctionRegistry[F_10_001_0213_01_0].eFunctionNumber                   := fbF_10_001_0213_01_0.ConfigFunction.eFunctionNumber; // Registration number


(****************************** 10-001-0213-02-0 ************************************)
(****************************** PalletMagazine Addon *************************************)
// Configuration function 
fbF_10_001_0213_02_0.ConfigFunction.FunctionName					:= '10-001-0213-02-0'; (* Function name *)
fbF_10_001_0213_02_0.ConfigFunction.eFunctionNumber				:= F_10_001_0213_02_0; (* Number of the function *)
fbF_10_001_0213_02_0.ConfigFunction.eFunctionType					:= E_FunctionType.NO_TYPE;
fbF_10_001_0213_02_0.ConfigFunction.eElementLink					:= E_ElementNumber.E_10_001_0213_00_0; 
fbF_10_001_0213_02_0.ConfigFunction.FunctionLink.eFunctionNumber	:= E_FunctionNumber.F_10_001_0213_01_0;	//Addon link to function, this is auto generated, an may need to be changed.
fbF_10_001_0213_02_0.ConfigFunction.FunctionLink.ZoneNumber		:= 1;		

fbF_10_001_0213_02_0.Config.TimeoutValueLift						:= T#20S; //Timeout when moving lift
fbF_10_001_0213_02_0.Config.TimeoutValueSeq						:= T#2M;  //Timeout for complete sequence
fbF_10_001_0213_02_0.Config.IdleStacking							:= FALSE; //Lift pallet up to optimze stacking

// Register function 
FunctionRegistry[F_10_001_0213_02_0].Enable                           := TRUE; (* Function will be called *)
FunctionRegistry[F_10_001_0213_02_0].eFunctionNumber                  := fbF_10_001_0213_02_0.ConfigFunction.eFunctionNumber; (* Registration number *)

(****************************** 10-001-0214-00-0 ************************************)
(*************************** ProBoxElement with one Motor *******************************)
// Configuration element 
fbEL_10_001_0214_00_0.ConfigElement.ElementName                     := '10-001-0214-00-0'; // Element name 
fbEL_10_001_0214_00_0.ConfigElement.eElementNumber                  := E_10_001_0214_00_0; // Number of the element 
fbEL_10_001_0214_00_0.ConfigElement.eSlaveElementNumber_34          := E_ElementNumber.E_BEGIN_ELEMENT; // Link from Master to slave element
fbEL_10_001_0214_00_0.ConfigElement.eElementType                    := E_ElementType.NO_TYPE; // No specific type

// Register element 
ElementRegistry[E_10_001_0214_00_0].Enable                          := TRUE; // Object is called
ElementRegistry[E_10_001_0214_00_0].eElementNumber                  := fbEL_10_001_0214_00_0.ConfigElement.eElementNumber; 

(****************************** 10-001-0214-01-0 ************************************)
(************************** ProBox Straight Transport *******************************)
// Configuration function
fbF_10_001_0214_01_0.ConfigFunction.FunctionName                       := '10-001-0214-01-0'; // Function name
fbF_10_001_0214_01_0.ConfigFunction.eFunctionNumber                    := F_10_001_0214_01_0; // Number of the function
fbF_10_001_0214_01_0.ConfigFunction.eElementLink                       := E_ElementNumber.E_10_001_0214_00_0;
fbF_10_001_0214_01_0.ConfigFunction.FunctionLink.eFunctionNumber       := E_FunctionNumber.F_BEGIN_FUNCTION;
fbF_10_001_0214_01_0.ConfigFunction.FunctionLink.ZoneNumber            := 0;
fbF_10_001_0214_01_0.ConfigFunction.eAdjacentFunctionNumberSide[1]     := E_FunctionNumber.F_10_001_0209_01_0;
fbF_10_001_0214_01_0.ConfigFunction.eAdjacentFunctionNumberSide[2]     := E_FunctionNumber.F_10_001_0215_01_0;
fbF_10_001_0214_01_0.ConfigFunction.ePrevFunctionNumber                := E_FunctionNumber.F_10_001_0209_01_0;
fbF_10_001_0214_01_0.ConfigFunction.eNextFunctionNumber                := E_FunctionNumber.F_10_001_0215_01_0;
fbF_10_001_0214_01_0.ConfigFunction.NumberOfZones                      := 1;
//Config zone 1
fbF_10_001_0214_01_0.ConfigFunction.Zone[1].ZoneName                   := '10-001-0214-01-1';
fbF_10_001_0214_01_0.ConfigFunction.Zone[1].EnableMFC                  := TRUE;
fbF_10_001_0214_01_0.ConfigFunction.Zone[1].EnableSimultaneousTransport:= FALSE; //Disable Simultaneous transport for multi zone functions
fbF_10_001_0214_01_0.ConfigFunction.Zone[1].EnableLatchOccupiedState   := TRUE;
fbF_10_001_0214_01_0.ConfigFunction.Zone[1].Length[1]                  := INT_TO_UINT(3000 / fbF_10_001_0214_01_0.ConfigFunction.NumberOfZones);	//Zone length (ie element length / number of zones)

// Register function
FunctionRegistry[F_10_001_0214_01_0].Enable                            := TRUE; (* Function will be called *)
FunctionRegistry[F_10_001_0214_01_0].eFunctionNumber                   := fbF_10_001_0214_01_0.ConfigFunction.eFunctionNumber; // Registration number


